Fanuc TP program (LS listing): FM203450.ls

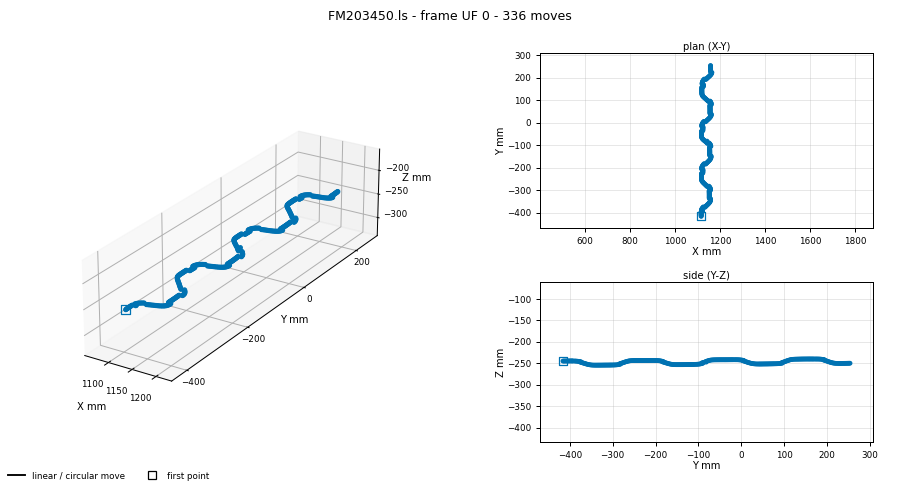
[picture p0: tool path of FM203450.ls in frame UF 0, 336 of 336 moves have a stored position in this frame; points joined in program order, loops and branches not executed]
/PROG  FM203450
/ATTR
OWNER		= MNEDITOR;
COMMENT		= "Auto FANUC move";
PROG_SIZE	= 0;
CREATE		= DATE 26-04-24  TIME 20:34:50;
MODIFIED	= DATE 26-04-24  TIME 20:34:50;
FILE_NAME	= ;
VERSION		= 0;
LINE_COUNT	= 341;
MEMORY_SIZE	= 0;
PROTECT		= READ_WRITE;
TCD:  STACK_SIZE	= 0,
      TASK_PRIORITY	= 50,
      TIME_SLICE	= 0,
      BUSY_LAMP_OFF	= 0,
      ABORT_REQUEST	= 0,
      PAUSE_REQUEST	= 0;
DEFAULT_GROUP	= 1,*,*,*,*;
CONTROL_CODE	= 00000000 00000000;
/MN
   1:  UFRAME_NUM=0 ;
   2:  UTOOL_NUM=1 ;
   3:  R[93]=10 ;
   4:  L P[1] 7mm/sec FINE ;
   5:  L P[2] 7mm/sec CNT50 ;
   6:  L P[3] 7mm/sec CNT50 ;
   7:  L P[4] 7mm/sec CNT50 ;
   8:  L P[5] 7mm/sec CNT50 ;
   9:  L P[6] 7mm/sec CNT50 ;
  10:  L P[7] 7mm/sec CNT50 ;
  11:  L P[8] 7mm/sec CNT50 ;
  12:  L P[9] 7mm/sec CNT50 ;
  13:  L P[10] 7mm/sec CNT50 ;
  14:  L P[11] 7mm/sec CNT50 ;
  15:  L P[12] 7mm/sec CNT50 ;
  16:  L P[13] 7mm/sec CNT50 ;
  17:  L P[14] 7mm/sec CNT50 ;
  18:  L P[15] 7mm/sec CNT50 ;
  19:  L P[16] 7mm/sec CNT50 ;
  20:  L P[17] 7mm/sec CNT50 ;
  21:  L P[18] 7mm/sec CNT50 ;
  22:  L P[19] 7mm/sec CNT50 ;
  23:  L P[20] 7mm/sec CNT50 ;
  24:  L P[21] 7mm/sec CNT50 ;
  25:  L P[22] 7mm/sec CNT50 ;
  26:  L P[23] 7mm/sec CNT50 ;
  27:  L P[24] 7mm/sec CNT50 ;
  28:  L P[25] 7mm/sec CNT50 ;
  29:  L P[26] 7mm/sec CNT50 ;
  30:  L P[27] 7mm/sec CNT50 ;
  31:  L P[28] 7mm/sec CNT50 ;
  32:  L P[29] 7mm/sec CNT50 ;
  33:  L P[30] 7mm/sec CNT50 ;
  34:  L P[31] 7mm/sec CNT50 ;
  35:  L P[32] 7mm/sec CNT50 ;
  36:  L P[33] 7mm/sec CNT50 ;
  37:  L P[34] 7mm/sec CNT50 ;
  38:  L P[35] 7mm/sec CNT50 ;
  39:  L P[36] 7mm/sec CNT50 ;
  40:  L P[37] 7mm/sec CNT50 ;
  41:  L P[38] 7mm/sec CNT50 ;
  42:  L P[39] 7mm/sec CNT50 ;
  43:  L P[40] 7mm/sec CNT50 ;
  44:  L P[41] 7mm/sec CNT50 ;
  45:  L P[42] 7mm/sec CNT50 ;
  46:  L P[43] 7mm/sec CNT50 ;
  47:  L P[44] 7mm/sec CNT50 ;
  48:  L P[45] 7mm/sec CNT50 ;
  49:  L P[46] 7mm/sec CNT50 ;
  50:  L P[47] 7mm/sec CNT50 ;
  51:  L P[48] 7mm/sec CNT50 ;
  52:  L P[49] 7mm/sec CNT50 ;
  53:  L P[50] 7mm/sec CNT50 ;
  54:  L P[51] 7mm/sec CNT50 ;
  55:  L P[52] 7mm/sec CNT50 ;
  56:  L P[53] 7mm/sec CNT50 ;
  57:  L P[54] 7mm/sec CNT50 ;
  58:  L P[55] 7mm/sec CNT50 ;
  59:  L P[56] 7mm/sec CNT50 ;
  60:  L P[57] 7mm/sec CNT50 ;
  61:  L P[58] 7mm/sec CNT50 ;
  62:  L P[59] 7mm/sec CNT50 ;
  63:  L P[60] 7mm/sec CNT50 ;
  64:  L P[61] 7mm/sec CNT50 ;
  65:  L P[62] 7mm/sec CNT50 ;
  66:  L P[63] 7mm/sec CNT50 ;
  67:  L P[64] 7mm/sec CNT50 ;
  68:  L P[65] 7mm/sec CNT50 ;
  69:  L P[66] 7mm/sec CNT50 ;
  70:  L P[67] 7mm/sec CNT50 ;
  71:  L P[68] 7mm/sec CNT50 ;
  72:  L P[69] 7mm/sec CNT50 ;
  73:  L P[70] 7mm/sec CNT50 ;
  74:  L P[71] 7mm/sec CNT50 ;
  75:  L P[72] 7mm/sec CNT50 ;
  76:  L P[73] 7mm/sec CNT50 ;
  77:  L P[74] 7mm/sec CNT50 ;
  78:  L P[75] 7mm/sec CNT50 ;
  79:  L P[76] 7mm/sec CNT50 ;
  80:  L P[77] 7mm/sec CNT50 ;
  81:  L P[78] 7mm/sec CNT50 ;
  82:  L P[79] 7mm/sec CNT50 ;
  83:  L P[80] 7mm/sec CNT50 ;
  84:  L P[81] 7mm/sec CNT50 ;
  85:  L P[82] 7mm/sec CNT50 ;
  86:  L P[83] 7mm/sec CNT50 ;
  87:  L P[84] 7mm/sec CNT50 ;
  88:  L P[85] 7mm/sec CNT50 ;
  89:  L P[86] 7mm/sec CNT50 ;
  90:  L P[87] 7mm/sec CNT50 ;
  91:  L P[88] 7mm/sec CNT50 ;
  92:  L P[89] 7mm/sec CNT50 ;
  93:  L P[90] 7mm/sec CNT50 ;
  94:  L P[91] 7mm/sec CNT50 ;
  95:  L P[92] 7mm/sec CNT50 ;
  96:  L P[93] 7mm/sec CNT50 ;
  97:  L P[94] 7mm/sec CNT50 ;
  98:  L P[95] 7mm/sec CNT50 ;
  99:  L P[96] 7mm/sec CNT50 ;
 100:  L P[97] 7mm/sec CNT50 ;
 101:  L P[98] 7mm/sec CNT50 ;
 102:  L P[99] 7mm/sec CNT50 ;
 103:  L P[100] 7mm/sec CNT50 ;
 104:  L P[101] 7mm/sec CNT50 ;
 105:  L P[102] 7mm/sec CNT50 ;
 106:  L P[103] 7mm/sec CNT50 ;
 107:  L P[104] 7mm/sec CNT50 ;
 108:  L P[105] 7mm/sec CNT50 ;
 109:  L P[106] 7mm/sec CNT50 ;
 110:  L P[107] 7mm/sec CNT50 ;
 111:  L P[108] 7mm/sec CNT50 ;
 112:  L P[109] 7mm/sec CNT50 ;
 113:  L P[110] 7mm/sec CNT50 ;
 114:  L P[111] 7mm/sec CNT50 ;
 115:  L P[112] 7mm/sec CNT50 ;
 116:  L P[113] 7mm/sec CNT50 ;
 117:  L P[114] 7mm/sec CNT50 ;
 118:  L P[115] 7mm/sec CNT50 ;
 119:  L P[116] 7mm/sec CNT50 ;
 120:  L P[117] 7mm/sec CNT50 ;
 121:  L P[118] 7mm/sec CNT50 ;
 122:  L P[119] 7mm/sec CNT50 ;
 123:  L P[120] 7mm/sec CNT50 ;
 124:  L P[121] 7mm/sec CNT50 ;
 125:  L P[122] 7mm/sec CNT50 ;
 126:  L P[123] 7mm/sec CNT50 ;
 127:  L P[124] 7mm/sec CNT50 ;
 128:  L P[125] 7mm/sec CNT50 ;
 129:  L P[126] 7mm/sec CNT50 ;
 130:  L P[127] 7mm/sec CNT50 ;
 131:  L P[128] 7mm/sec CNT50 ;
 132:  L P[129] 7mm/sec CNT50 ;
 133:  L P[130] 7mm/sec CNT50 ;
 134:  L P[131] 7mm/sec CNT50 ;
 135:  L P[132] 7mm/sec CNT50 ;
 136:  L P[133] 7mm/sec CNT50 ;
 137:  L P[134] 7mm/sec CNT50 ;
 138:  L P[135] 7mm/sec CNT50 ;
 139:  L P[136] 7mm/sec CNT50 ;
 140:  L P[137] 7mm/sec CNT50 ;
 141:  L P[138] 7mm/sec CNT50 ;
 142:  L P[139] 7mm/sec CNT50 ;
 143:  L P[140] 7mm/sec CNT50 ;
 144:  L P[141] 7mm/sec CNT50 ;
 145:  L P[142] 7mm/sec CNT50 ;
 146:  L P[143] 7mm/sec CNT50 ;
 147:  L P[144] 7mm/sec CNT50 ;
 148:  L P[145] 7mm/sec CNT50 ;
 149:  L P[146] 7mm/sec CNT50 ;
 150:  L P[147] 7mm/sec CNT50 ;
 151:  L P[148] 7mm/sec CNT50 ;
 152:  L P[149] 7mm/sec CNT50 ;
 153:  L P[150] 7mm/sec CNT50 ;
 154:  L P[151] 7mm/sec CNT50 ;
 155:  L P[152] 7mm/sec CNT50 ;
 156:  L P[153] 7mm/sec CNT50 ;
 157:  L P[154] 7mm/sec CNT50 ;
 158:  L P[155] 7mm/sec CNT50 ;
 159:  L P[156] 7mm/sec CNT50 ;
 160:  L P[157] 7mm/sec CNT50 ;
 161:  L P[158] 7mm/sec CNT50 ;
 162:  L P[159] 7mm/sec CNT50 ;
 163:  L P[160] 7mm/sec CNT50 ;
 164:  L P[161] 7mm/sec CNT50 ;
 165:  L P[162] 7mm/sec CNT50 ;
 166:  L P[163] 7mm/sec CNT50 ;
 167:  L P[164] 7mm/sec CNT50 ;
 168:  L P[165] 7mm/sec CNT50 ;
 169:  L P[166] 7mm/sec CNT50 ;
 170:  L P[167] 7mm/sec CNT50 ;
 171:  L P[168] 7mm/sec CNT50 ;
 172:  L P[169] 7mm/sec CNT50 ;
 173:  L P[170] 7mm/sec CNT50 ;
 174:  L P[171] 7mm/sec CNT50 ;
 175:  L P[172] 7mm/sec CNT50 ;
 176:  L P[173] 7mm/sec CNT50 ;
 177:  L P[174] 7mm/sec CNT50 ;
 178:  L P[175] 7mm/sec CNT50 ;
 179:  L P[176] 7mm/sec CNT50 ;
 180:  L P[177] 7mm/sec CNT50 ;
 181:  L P[178] 7mm/sec CNT50 ;
 182:  L P[179] 7mm/sec CNT50 ;
 183:  L P[180] 7mm/sec CNT50 ;
 184:  L P[181] 7mm/sec CNT50 ;
 185:  L P[182] 7mm/sec CNT50 ;
 186:  L P[183] 7mm/sec CNT50 ;
 187:  L P[184] 7mm/sec CNT50 ;
 188:  L P[185] 7mm/sec CNT50 ;
 189:  L P[186] 7mm/sec CNT50 ;
 190:  L P[187] 7mm/sec CNT50 ;
 191:  L P[188] 7mm/sec CNT50 ;
 192:  L P[189] 7mm/sec CNT50 ;
 193:  L P[190] 7mm/sec CNT50 ;
 194:  L P[191] 7mm/sec CNT50 ;
 195:  L P[192] 7mm/sec CNT50 ;
 196:  L P[193] 7mm/sec CNT50 ;
 197:  L P[194] 7mm/sec CNT50 ;
 198:  L P[195] 7mm/sec CNT50 ;
 199:  L P[196] 7mm/sec CNT50 ;
 200:  L P[197] 7mm/sec CNT50 ;
 201:  L P[198] 7mm/sec CNT50 ;
 202:  L P[199] 7mm/sec CNT50 ;
 203:  L P[200] 7mm/sec CNT50 ;
 204:  L P[201] 7mm/sec CNT50 ;
 205:  L P[202] 7mm/sec CNT50 ;
 206:  L P[203] 7mm/sec CNT50 ;
 207:  L P[204] 7mm/sec CNT50 ;
 208:  L P[205] 7mm/sec CNT50 ;
 209:  L P[206] 7mm/sec CNT50 ;
 210:  L P[207] 7mm/sec CNT50 ;
 211:  L P[208] 7mm/sec CNT50 ;
 212:  L P[209] 7mm/sec CNT50 ;
 213:  L P[210] 7mm/sec CNT50 ;
 214:  L P[211] 7mm/sec CNT50 ;
 215:  L P[212] 7mm/sec CNT50 ;
 216:  L P[213] 7mm/sec CNT50 ;
 217:  L P[214] 7mm/sec CNT50 ;
 218:  L P[215] 7mm/sec CNT50 ;
 219:  L P[216] 7mm/sec CNT50 ;
 220:  L P[217] 7mm/sec CNT50 ;
 221:  L P[218] 7mm/sec CNT50 ;
 222:  L P[219] 7mm/sec CNT50 ;
 223:  L P[220] 7mm/sec CNT50 ;
 224:  L P[221] 7mm/sec CNT50 ;
 225:  L P[222] 7mm/sec CNT50 ;
 226:  L P[223] 7mm/sec CNT50 ;
 227:  L P[224] 7mm/sec CNT50 ;
 228:  L P[225] 7mm/sec CNT50 ;
 229:  L P[226] 7mm/sec CNT50 ;
 230:  L P[227] 7mm/sec CNT50 ;
 231:  L P[228] 7mm/sec CNT50 ;
 232:  L P[229] 7mm/sec CNT50 ;
 233:  L P[230] 7mm/sec CNT50 ;
 234:  L P[231] 7mm/sec CNT50 ;
 235:  L P[232] 7mm/sec CNT50 ;
 236:  L P[233] 7mm/sec CNT50 ;
 237:  L P[234] 7mm/sec CNT50 ;
 238:  L P[235] 7mm/sec CNT50 ;
 239:  L P[236] 7mm/sec CNT50 ;
 240:  L P[237] 7mm/sec CNT50 ;
 241:  L P[238] 7mm/sec CNT50 ;
 242:  L P[239] 7mm/sec CNT50 ;
 243:  L P[240] 7mm/sec CNT50 ;
 244:  L P[241] 7mm/sec CNT50 ;
 245:  L P[242] 7mm/sec CNT50 ;
 246:  L P[243] 7mm/sec CNT50 ;
 247:  L P[244] 7mm/sec CNT50 ;
 248:  L P[245] 7mm/sec CNT50 ;
 249:  L P[246] 7mm/sec CNT50 ;
 250:  L P[247] 7mm/sec CNT50 ;
 251:  L P[248] 7mm/sec CNT50 ;
 252:  L P[249] 7mm/sec CNT50 ;
 253:  L P[250] 7mm/sec CNT50 ;
 254:  L P[251] 7mm/sec CNT50 ;
 255:  L P[252] 7mm/sec CNT50 ;
 256:  L P[253] 7mm/sec CNT50 ;
 257:  L P[254] 7mm/sec CNT50 ;
 258:  L P[255] 7mm/sec CNT50 ;
 259:  L P[256] 7mm/sec CNT50 ;
 260:  L P[257] 7mm/sec CNT50 ;
 261:  L P[258] 7mm/sec CNT50 ;
 262:  L P[259] 7mm/sec CNT50 ;
 263:  L P[260] 7mm/sec CNT50 ;
 264:  L P[261] 7mm/sec CNT50 ;
 265:  L P[262] 7mm/sec CNT50 ;
 266:  L P[263] 7mm/sec CNT50 ;
 267:  L P[264] 7mm/sec CNT50 ;
 268:  L P[265] 7mm/sec CNT50 ;
 269:  L P[266] 7mm/sec CNT50 ;
 270:  L P[267] 7mm/sec CNT50 ;
 271:  L P[268] 7mm/sec CNT50 ;
 272:  L P[269] 7mm/sec CNT50 ;
 273:  L P[270] 7mm/sec CNT50 ;
 274:  L P[271] 7mm/sec CNT50 ;
 275:  L P[272] 7mm/sec CNT50 ;
 276:  L P[273] 7mm/sec CNT50 ;
 277:  L P[274] 7mm/sec CNT50 ;
 278:  L P[275] 7mm/sec CNT50 ;
 279:  L P[276] 7mm/sec CNT50 ;
 280:  L P[277] 7mm/sec CNT50 ;
 281:  L P[278] 7mm/sec CNT50 ;
 282:  L P[279] 7mm/sec CNT50 ;
 283:  L P[280] 7mm/sec CNT50 ;
 284:  L P[281] 7mm/sec CNT50 ;
 285:  L P[282] 7mm/sec CNT50 ;
 286:  L P[283] 7mm/sec CNT50 ;
 287:  L P[284] 7mm/sec CNT50 ;
 288:  L P[285] 7mm/sec CNT50 ;
 289:  L P[286] 7mm/sec CNT50 ;
 290:  L P[287] 7mm/sec CNT50 ;
 291:  L P[288] 7mm/sec CNT50 ;
 292:  L P[289] 7mm/sec CNT50 ;
 293:  L P[290] 7mm/sec CNT50 ;
 294:  L P[291] 7mm/sec CNT50 ;
 295:  L P[292] 7mm/sec CNT50 ;
 296:  L P[293] 7mm/sec CNT50 ;
 297:  L P[294] 7mm/sec CNT50 ;
 298:  L P[295] 7mm/sec CNT50 ;
 299:  L P[296] 7mm/sec CNT50 ;
 300:  L P[297] 7mm/sec CNT50 ;
 301:  L P[298] 7mm/sec CNT50 ;
 302:  L P[299] 7mm/sec CNT50 ;
 303:  L P[300] 7mm/sec CNT50 ;
 304:  L P[301] 7mm/sec CNT50 ;
 305:  L P[302] 7mm/sec CNT50 ;
 306:  L P[303] 7mm/sec CNT50 ;
 307:  L P[304] 7mm/sec CNT50 ;
 308:  L P[305] 7mm/sec CNT50 ;
 309:  L P[306] 7mm/sec CNT50 ;
 310:  L P[307] 7mm/sec CNT50 ;
 311:  L P[308] 7mm/sec CNT50 ;
 312:  L P[309] 7mm/sec CNT50 ;
 313:  L P[310] 7mm/sec CNT50 ;
 314:  L P[311] 7mm/sec CNT50 ;
 315:  L P[312] 7mm/sec CNT50 ;
 316:  L P[313] 7mm/sec CNT50 ;
 317:  L P[314] 7mm/sec CNT50 ;
 318:  L P[315] 7mm/sec CNT50 ;
 319:  L P[316] 7mm/sec CNT50 ;
 320:  L P[317] 7mm/sec CNT50 ;
 321:  L P[318] 7mm/sec CNT50 ;
 322:  L P[319] 7mm/sec CNT50 ;
 323:  L P[320] 7mm/sec CNT50 ;
 324:  L P[321] 7mm/sec CNT50 ;
 325:  L P[322] 7mm/sec CNT50 ;
 326:  L P[323] 7mm/sec CNT50 ;
 327:  L P[324] 7mm/sec CNT50 ;
 328:  L P[325] 7mm/sec CNT50 ;
 329:  L P[326] 7mm/sec CNT50 ;
 330:  L P[327] 7mm/sec CNT50 ;
 331:  L P[328] 7mm/sec CNT50 ;
 332:  L P[329] 7mm/sec CNT50 ;
 333:  L P[330] 7mm/sec CNT50 ;
 334:  L P[331] 7mm/sec CNT50 ;
 335:  L P[332] 7mm/sec CNT50 ;
 336:  L P[333] 7mm/sec CNT50 ;
 337:  L P[334] 7mm/sec CNT50 ;
 338:  L P[335] 7mm/sec CNT50 ;
 339:  L P[336] 7mm/sec FINE ;
 340:  R[93]=1 ;
 341:  END ;
/POS
P[1]{
   GP1:
	UF : 0, UT : 1,		CONFIG : 'N U T, 0, 0, 0',
	X = 1117.238  mm,	Y = -416.121  mm,	Z = -244.812  mm,
	W = 0.000 deg,	P = 30.000 deg,	R = 175.456 deg
};
P[2]{
   GP1:
	UF : 0, UT : 1,		CONFIG : 'N U T, 0, 0, 0',
	X = 1117.157  mm,	Y = -414.122  mm,	Z = -244.780  mm,
	W = 0.000 deg,	P = 30.000 deg,	R = 175.456 deg
};
P[3]{
   GP1:
	UF : 0, UT : 1,		CONFIG : 'N U T, 0, 0, 0',
	X = 1117.075  mm,	Y = -412.113  mm,	Z = -244.742  mm,
	W = 0.000 deg,	P = 30.000 deg,	R = 175.456 deg
};
P[4]{
   GP1:
	UF : 0, UT : 1,		CONFIG : 'N U T, 0, 0, 0',
	X = 1117.006  mm,	Y = -410.100  mm,	Z = -244.707  mm,
	W = 0.000 deg,	P = 30.000 deg,	R = 175.456 deg
};
P[5]{
   GP1:
	UF : 0, UT : 1,		CONFIG : 'N U T, 0, 0, 0',
	X = 1116.940  mm,	Y = -408.081  mm,	Z = -244.666  mm,
	W = 0.000 deg,	P = 30.000 deg,	R = 175.456 deg
};
P[6]{
   GP1:
	UF : 0, UT : 1,		CONFIG : 'N U T, 0, 0, 0',
	X = 1116.897  mm,	Y = -406.053  mm,	Z = -244.628  mm,
	W = 0.000 deg,	P = 30.000 deg,	R = 175.456 deg
};
P[7]{
   GP1:
	UF : 0, UT : 1,		CONFIG : 'N U T, 0, 0, 0',
	X = 1116.868  mm,	Y = -404.029  mm,	Z = -244.597  mm,
	W = 0.000 deg,	P = 30.000 deg,	R = 175.456 deg
};
P[8]{
   GP1:
	UF : 0, UT : 1,		CONFIG : 'N U T, 0, 0, 0',
	X = 1116.858  mm,	Y = -402.004  mm,	Z = -244.573  mm,
	W = 0.000 deg,	P = 30.000 deg,	R = 175.456 deg
};
P[9]{
   GP1:
	UF : 0, UT : 1,		CONFIG : 'N U T, 0, 0, 0',
	X = 1116.863  mm,	Y = -399.971  mm,	Z = -244.558  mm,
	W = 0.000 deg,	P = 30.000 deg,	R = 175.456 deg
};
P[10]{
   GP1:
	UF : 0, UT : 1,		CONFIG : 'N U T, 0, 0, 0',
	X = 1116.898  mm,	Y = -397.917  mm,	Z = -244.550  mm,
	W = 0.000 deg,	P = 30.000 deg,	R = 175.456 deg
};
P[11]{
   GP1:
	UF : 0, UT : 1,		CONFIG : 'N U T, 0, 0, 0',
	X = 1116.977  mm,	Y = -395.859  mm,	Z = -244.552  mm,
	W = 0.000 deg,	P = 30.000 deg,	R = 175.456 deg
};
P[12]{
   GP1:
	UF : 0, UT : 1,		CONFIG : 'N U T, 0, 0, 0',
	X = 1123.071  mm,	Y = -394.287  mm,	Z = -244.568  mm,
	W = 0.000 deg,	P = 30.000 deg,	R = 175.456 deg
};
P[13]{
   GP1:
	UF : 0, UT : 1,		CONFIG : 'N U T, 0, 0, 0',
	X = 1123.311  mm,	Y = -392.534  mm,	Z = -244.620  mm,
	W = 0.000 deg,	P = 30.000 deg,	R = 170.071 deg
};
P[14]{
   GP1:
	UF : 0, UT : 1,		CONFIG : 'N U T, 0, 0, 0',
	X = 1117.902  mm,	Y = -389.257  mm,	Z = -244.722  mm,
	W = 0.000 deg,	P = 30.000 deg,	R = 162.234 deg
};
P[15]{
   GP1:
	UF : 0, UT : 1,		CONFIG : 'N U T, 0, 0, 0',
	X = 1118.551  mm,	Y = -387.006  mm,	Z = -244.847  mm,
	W = 0.000 deg,	P = 30.000 deg,	R = 154.276 deg
};
P[16]{
   GP1:
	UF : 0, UT : 1,		CONFIG : 'N U T, 0, 0, 0',
	X = 1119.505  mm,	Y = -384.707  mm,	Z = -245.002  mm,
	W = 0.000 deg,	P = 30.000 deg,	R = 145.985 deg
};
P[17]{
   GP1:
	UF : 0, UT : 1,		CONFIG : 'N U T, 0, 0, 0',
	X = 1120.698  mm,	Y = -382.492  mm,	Z = -245.205  mm,
	W = 0.000 deg,	P = 30.000 deg,	R = 137.274 deg
};
P[18]{
   GP1:
	UF : 0, UT : 1,		CONFIG : 'N U T, 0, 0, 0',
	X = 1122.055  mm,	Y = -380.317  mm,	Z = -245.479  mm,
	W = 0.000 deg,	P = 30.000 deg,	R = 137.274 deg
};
P[19]{
   GP1:
	UF : 0, UT : 1,		CONFIG : 'N U T, 0, 0, 0',
	X = 1123.594  mm,	Y = -378.210  mm,	Z = -245.828  mm,
	W = 0.000 deg,	P = 30.000 deg,	R = 137.274 deg
};
P[20]{
   GP1:
	UF : 0, UT : 1,		CONFIG : 'N U T, 0, 0, 0',
	X = 1125.169  mm,	Y = -376.126  mm,	Z = -246.227  mm,
	W = 0.000 deg,	P = 30.000 deg,	R = 137.274 deg
};
P[21]{
   GP1:
	UF : 0, UT : 1,		CONFIG : 'N U T, 0, 0, 0',
	X = 1126.962  mm,	Y = -374.005  mm,	Z = -246.664  mm,
	W = 0.000 deg,	P = 30.000 deg,	R = 137.274 deg
};
P[22]{
   GP1:
	UF : 0, UT : 1,		CONFIG : 'N U T, 0, 0, 0',
	X = 1133.263  mm,	Y = -376.051  mm,	Z = -247.177  mm,
	W = 0.000 deg,	P = 30.000 deg,	R = 137.274 deg
};
P[23]{
   GP1:
	UF : 0, UT : 1,		CONFIG : 'N U T, 0, 0, 0',
	X = 1135.120  mm,	Y = -374.071  mm,	Z = -247.739  mm,
	W = 0.000 deg,	P = 30.000 deg,	R = 137.274 deg
};
P[24]{
   GP1:
	UF : 0, UT : 1,		CONFIG : 'N U T, 0, 0, 0',
	X = 1137.025  mm,	Y = -372.109  mm,	Z = -248.355  mm,
	W = 0.000 deg,	P = 30.000 deg,	R = 137.274 deg
};
P[25]{
   GP1:
	UF : 0, UT : 1,		CONFIG : 'N U T, 0, 0, 0',
	X = 1138.998  mm,	Y = -370.148  mm,	Z = -248.981  mm,
	W = 0.000 deg,	P = 30.000 deg,	R = 137.274 deg
};
P[26]{
   GP1:
	UF : 0, UT : 1,		CONFIG : 'N U T, 0, 0, 0',
	X = 1141.067  mm,	Y = -368.170  mm,	Z = -249.617  mm,
	W = 0.000 deg,	P = 30.000 deg,	R = 137.274 deg
};
P[27]{
   GP1:
	UF : 0, UT : 1,		CONFIG : 'N U T, 0, 0, 0',
	X = 1143.185  mm,	Y = -366.152  mm,	Z = -250.236  mm,
	W = 0.000 deg,	P = 30.000 deg,	R = 137.274 deg
};
P[28]{
   GP1:
	UF : 0, UT : 1,		CONFIG : 'N U T, 0, 0, 0',
	X = 1145.220  mm,	Y = -364.138  mm,	Z = -250.854  mm,
	W = 0.000 deg,	P = 30.000 deg,	R = 137.274 deg
};
P[29]{
   GP1:
	UF : 0, UT : 1,		CONFIG : 'N U T, 0, 0, 0',
	X = 1147.260  mm,	Y = -362.140  mm,	Z = -251.461  mm,
	W = 0.000 deg,	P = 30.000 deg,	R = 143.931 deg
};
P[30]{
   GP1:
	UF : 0, UT : 1,		CONFIG : 'N U T, 0, 0, 0',
	X = 1149.327  mm,	Y = -360.100  mm,	Z = -252.059  mm,
	W = 0.000 deg,	P = 30.000 deg,	R = 156.053 deg
};
P[31]{
   GP1:
	UF : 0, UT : 1,		CONFIG : 'N U T, 0, 0, 0',
	X = 1151.305  mm,	Y = -358.012  mm,	Z = -252.604  mm,
	W = 0.000 deg,	P = 30.000 deg,	R = 167.750 deg
};
P[32]{
   GP1:
	UF : 0, UT : 1,		CONFIG : 'N U T, 0, 0, 0',
	X = 1153.153  mm,	Y = -355.863  mm,	Z = -253.093  mm,
	W = 0.000 deg,	P = 30.000 deg,	R = 178.930 deg
};
P[33]{
   GP1:
	UF : 0, UT : 1,		CONFIG : 'N U T, 0, 0, 0',
	X = 1154.738  mm,	Y = -353.672  mm,	Z = -253.493  mm,
	W = 0.000 deg,	P = 30.000 deg,	R = 178.930 deg
};
P[34]{
   GP1:
	UF : 0, UT : 1,		CONFIG : 'N U T, 0, 0, 0',
	X = 1156.111  mm,	Y = -351.454  mm,	Z = -253.825  mm,
	W = 0.000 deg,	P = 30.000 deg,	R = 178.930 deg
};
P[35]{
   GP1:
	UF : 0, UT : 1,		CONFIG : 'N U T, 0, 0, 0',
	X = 1157.241  mm,	Y = -349.136  mm,	Z = -254.072  mm,
	W = 0.000 deg,	P = 30.000 deg,	R = 178.930 deg
};
P[36]{
   GP1:
	UF : 0, UT : 1,		CONFIG : 'N U T, 0, 0, 0',
	X = 1158.022  mm,	Y = -346.774  mm,	Z = -254.230  mm,
	W = 0.000 deg,	P = 30.000 deg,	R = 178.930 deg
};
P[37]{
   GP1:
	UF : 0, UT : 1,		CONFIG : 'N U T, 0, 0, 0',
	X = 1158.497  mm,	Y = -344.458  mm,	Z = -254.317  mm,
	W = 0.000 deg,	P = 30.000 deg,	R = 178.930 deg
};
P[38]{
   GP1:
	UF : 0, UT : 1,		CONFIG : 'N U T, 0, 0, 0',
	X = 1158.732  mm,	Y = -342.235  mm,	Z = -254.352  mm,
	W = 0.000 deg,	P = 30.000 deg,	R = 178.930 deg
};
P[39]{
   GP1:
	UF : 0, UT : 1,		CONFIG : 'N U T, 0, 0, 0',
	X = 1158.843  mm,	Y = -340.119  mm,	Z = -254.355  mm,
	W = 0.000 deg,	P = 30.000 deg,	R = 178.930 deg
};
P[40]{
   GP1:
	UF : 0, UT : 1,		CONFIG : 'N U T, 0, 0, 0',
	X = 1158.899  mm,	Y = -338.073  mm,	Z = -254.354  mm,
	W = 0.000 deg,	P = 30.000 deg,	R = 178.930 deg
};
P[41]{
   GP1:
	UF : 0, UT : 1,		CONFIG : 'N U T, 0, 0, 0',
	X = 1152.944  mm,	Y = -335.946  mm,	Z = -254.352  mm,
	W = 0.000 deg,	P = 30.000 deg,	R = 178.930 deg
};
P[42]{
   GP1:
	UF : 0, UT : 1,		CONFIG : 'N U T, 0, 0, 0',
	X = 1152.971  mm,	Y = -333.966  mm,	Z = -254.346  mm,
	W = 0.000 deg,	P = 30.000 deg,	R = 178.930 deg
};
P[43]{
   GP1:
	UF : 0, UT : 1,		CONFIG : 'N U T, 0, 0, 0',
	X = 1152.989  mm,	Y = -331.976  mm,	Z = -254.338  mm,
	W = 0.000 deg,	P = 30.000 deg,	R = 178.930 deg
};
P[44]{
   GP1:
	UF : 0, UT : 1,		CONFIG : 'N U T, 0, 0, 0',
	X = 1153.003  mm,	Y = -329.982  mm,	Z = -254.324  mm,
	W = 0.000 deg,	P = 30.000 deg,	R = 178.930 deg
};
P[45]{
   GP1:
	UF : 0, UT : 1,		CONFIG : 'N U T, 0, 0, 0',
	X = 1153.013  mm,	Y = -327.989  mm,	Z = -254.307  mm,
	W = 0.000 deg,	P = 30.000 deg,	R = 178.930 deg
};
P[46]{
   GP1:
	UF : 0, UT : 1,		CONFIG : 'N U T, 0, 0, 0',
	X = 1153.018  mm,	Y = -325.995  mm,	Z = -254.288  mm,
	W = 0.000 deg,	P = 30.000 deg,	R = 178.930 deg
};
P[47]{
   GP1:
	UF : 0, UT : 1,		CONFIG : 'N U T, 0, 0, 0',
	X = 1153.020  mm,	Y = -323.998  mm,	Z = -254.268  mm,
	W = 0.000 deg,	P = 30.000 deg,	R = 178.930 deg
};
P[48]{
   GP1:
	UF : 0, UT : 1,		CONFIG : 'N U T, 0, 0, 0',
	X = 1153.020  mm,	Y = -322.002  mm,	Z = -254.247  mm,
	W = 0.000 deg,	P = 30.000 deg,	R = 178.930 deg
};
P[49]{
   GP1:
	UF : 0, UT : 1,		CONFIG : 'N U T, 0, 0, 0',
	X = 1153.017  mm,	Y = -320.009  mm,	Z = -254.228  mm,
	W = 0.000 deg,	P = 30.000 deg,	R = 178.930 deg
};
P[50]{
   GP1:
	UF : 0, UT : 1,		CONFIG : 'N U T, 0, 0, 0',
	X = 1153.008  mm,	Y = -318.019  mm,	Z = -254.209  mm,
	W = 0.000 deg,	P = 30.000 deg,	R = 178.930 deg
};
P[51]{
   GP1:
	UF : 0, UT : 1,		CONFIG : 'N U T, 0, 0, 0',
	X = 1152.993  mm,	Y = -316.026  mm,	Z = -254.195  mm,
	W = 0.000 deg,	P = 30.000 deg,	R = 178.930 deg
};
P[52]{
   GP1:
	UF : 0, UT : 1,		CONFIG : 'N U T, 0, 0, 0',
	X = 1152.973  mm,	Y = -314.036  mm,	Z = -254.181  mm,
	W = 0.000 deg,	P = 30.000 deg,	R = 178.930 deg
};
P[53]{
   GP1:
	UF : 0, UT : 1,		CONFIG : 'N U T, 0, 0, 0',
	X = 1152.945  mm,	Y = -312.050  mm,	Z = -254.166  mm,
	W = 0.000 deg,	P = 30.000 deg,	R = 178.930 deg
};
P[54]{
   GP1:
	UF : 0, UT : 1,		CONFIG : 'N U T, 0, 0, 0',
	X = 1152.907  mm,	Y = -310.067  mm,	Z = -254.149  mm,
	W = 0.000 deg,	P = 30.000 deg,	R = 178.930 deg
};
P[55]{
   GP1:
	UF : 0, UT : 1,		CONFIG : 'N U T, 0, 0, 0',
	X = 1152.856  mm,	Y = -308.083  mm,	Z = -254.127  mm,
	W = 0.000 deg,	P = 30.000 deg,	R = 178.930 deg
};
P[56]{
   GP1:
	UF : 0, UT : 1,		CONFIG : 'N U T, 0, 0, 0',
	X = 1152.797  mm,	Y = -306.094  mm,	Z = -254.104  mm,
	W = 0.000 deg,	P = 30.000 deg,	R = 178.930 deg
};
P[57]{
   GP1:
	UF : 0, UT : 1,		CONFIG : 'N U T, 0, 0, 0',
	X = 1152.731  mm,	Y = -304.105  mm,	Z = -254.075  mm,
	W = 0.000 deg,	P = 30.000 deg,	R = 178.930 deg
};
P[58]{
   GP1:
	UF : 0, UT : 1,		CONFIG : 'N U T, 0, 0, 0',
	X = 1152.659  mm,	Y = -302.140  mm,	Z = -254.045  mm,
	W = 0.000 deg,	P = 30.000 deg,	R = 178.930 deg
};
P[59]{
   GP1:
	UF : 0, UT : 1,		CONFIG : 'N U T, 0, 0, 0',
	X = 1158.536  mm,	Y = -299.819  mm,	Z = -253.999  mm,
	W = 0.000 deg,	P = 30.000 deg,	R = -172.792 deg
};
P[60]{
   GP1:
	UF : 0, UT : 1,		CONFIG : 'N U T, 0, 0, 0',
	X = 1158.403  mm,	Y = -297.754  mm,	Z = -253.948  mm,
	W = 0.000 deg,	P = 30.000 deg,	R = -163.956 deg
};
P[61]{
   GP1:
	UF : 0, UT : 1,		CONFIG : 'N U T, 0, 0, 0',
	X = 1158.189  mm,	Y = -295.627  mm,	Z = -253.878  mm,
	W = 0.000 deg,	P = 30.000 deg,	R = -155.091 deg
};
P[62]{
   GP1:
	UF : 0, UT : 1,		CONFIG : 'N U T, 0, 0, 0',
	X = 1157.847  mm,	Y = -293.378  mm,	Z = -253.781  mm,
	W = 0.000 deg,	P = 30.000 deg,	R = -146.168 deg
};
P[63]{
   GP1:
	UF : 0, UT : 1,		CONFIG : 'N U T, 0, 0, 0',
	X = 1157.172  mm,	Y = -290.942  mm,	Z = -253.605  mm,
	W = 0.000 deg,	P = 30.000 deg,	R = -136.996 deg
};
P[64]{
   GP1:
	UF : 0, UT : 1,		CONFIG : 'N U T, 0, 0, 0',
	X = 1156.021  mm,	Y = -288.532  mm,	Z = -253.312  mm,
	W = 0.000 deg,	P = 30.000 deg,	R = -136.996 deg
};
P[65]{
   GP1:
	UF : 0, UT : 1,		CONFIG : 'N U T, 0, 0, 0',
	X = 1154.591  mm,	Y = -286.300  mm,	Z = -252.918  mm,
	W = 0.000 deg,	P = 30.000 deg,	R = -136.996 deg
};
P[66]{
   GP1:
	UF : 0, UT : 1,		CONFIG : 'N U T, 0, 0, 0',
	X = 1152.986  mm,	Y = -284.113  mm,	Z = -252.468  mm,
	W = 0.000 deg,	P = 30.000 deg,	R = -136.996 deg
};
P[67]{
   GP1:
	UF : 0, UT : 1,		CONFIG : 'N U T, 0, 0, 0',
	X = 1151.105  mm,	Y = -281.983  mm,	Z = -251.928  mm,
	W = 0.000 deg,	P = 30.000 deg,	R = -136.996 deg
};
P[68]{
   GP1:
	UF : 0, UT : 1,		CONFIG : 'N U T, 0, 0, 0',
	X = 1144.899  mm,	Y = -284.123  mm,	Z = -251.352  mm,
	W = 0.000 deg,	P = 30.000 deg,	R = -136.996 deg
};
P[69]{
   GP1:
	UF : 0, UT : 1,		CONFIG : 'N U T, 0, 0, 0',
	X = 1142.839  mm,	Y = -282.199  mm,	Z = -250.685  mm,
	W = 0.000 deg,	P = 30.000 deg,	R = -136.996 deg
};
P[70]{
   GP1:
	UF : 0, UT : 1,		CONFIG : 'N U T, 0, 0, 0',
	X = 1140.618  mm,	Y = -280.151  mm,	Z = -250.008  mm,
	W = 0.000 deg,	P = 30.000 deg,	R = -136.996 deg
};
P[71]{
   GP1:
	UF : 0, UT : 1,		CONFIG : 'N U T, 0, 0, 0',
	X = 1138.641  mm,	Y = -278.119  mm,	Z = -249.386  mm,
	W = 0.000 deg,	P = 30.000 deg,	R = -136.996 deg
};
P[72]{
   GP1:
	UF : 0, UT : 1,		CONFIG : 'N U T, 0, 0, 0',
	X = 1136.600  mm,	Y = -276.125  mm,	Z = -248.711  mm,
	W = 0.000 deg,	P = 30.000 deg,	R = -136.996 deg
};
P[73]{
   GP1:
	UF : 0, UT : 1,		CONFIG : 'N U T, 0, 0, 0',
	X = 1134.609  mm,	Y = -274.102  mm,	Z = -248.054  mm,
	W = 0.000 deg,	P = 30.000 deg,	R = -136.996 deg
};
P[74]{
   GP1:
	UF : 0, UT : 1,		CONFIG : 'N U T, 0, 0, 0',
	X = 1132.747  mm,	Y = -272.196  mm,	Z = -247.379  mm,
	W = 0.000 deg,	P = 30.000 deg,	R = -136.996 deg
};
P[75]{
   GP1:
	UF : 0, UT : 1,		CONFIG : 'N U T, 0, 0, 0',
	X = 1130.424  mm,	Y = -270.212  mm,	Z = -246.656  mm,
	W = 0.000 deg,	P = 30.000 deg,	R = -136.996 deg
};
P[76]{
   GP1:
	UF : 0, UT : 1,		CONFIG : 'N U T, 0, 0, 0',
	X = 1128.315  mm,	Y = -268.134  mm,	Z = -246.043  mm,
	W = 0.000 deg,	P = 30.000 deg,	R = -144.486 deg
};
P[77]{
   GP1:
	UF : 0, UT : 1,		CONFIG : 'N U T, 0, 0, 0',
	X = 1126.263  mm,	Y = -266.105  mm,	Z = -245.449  mm,
	W = 0.000 deg,	P = 30.000 deg,	R = -157.136 deg
};
P[78]{
   GP1:
	UF : 0, UT : 1,		CONFIG : 'N U T, 0, 0, 0',
	X = 1124.213  mm,	Y = -263.958  mm,	Z = -244.899  mm,
	W = 0.000 deg,	P = 30.000 deg,	R = -169.430 deg
};
P[79]{
   GP1:
	UF : 0, UT : 1,		CONFIG : 'N U T, 0, 0, 0',
	X = 1122.535  mm,	Y = -261.771  mm,	Z = -244.489  mm,
	W = 0.000 deg,	P = 30.000 deg,	R = 179.462 deg
};
P[80]{
   GP1:
	UF : 0, UT : 1,		CONFIG : 'N U T, 0, 0, 0',
	X = 1121.010  mm,	Y = -259.579  mm,	Z = -244.131  mm,
	W = 0.000 deg,	P = 30.000 deg,	R = 179.462 deg
};
P[81]{
   GP1:
	UF : 0, UT : 1,		CONFIG : 'N U T, 0, 0, 0',
	X = 1119.695  mm,	Y = -257.117  mm,	Z = -243.885  mm,
	W = 0.000 deg,	P = 30.000 deg,	R = 179.462 deg
};
P[82]{
   GP1:
	UF : 0, UT : 1,		CONFIG : 'N U T, 0, 0, 0',
	X = 1119.040  mm,	Y = -254.711  mm,	Z = -243.744  mm,
	W = 0.000 deg,	P = 30.000 deg,	R = 179.462 deg
};
P[83]{
   GP1:
	UF : 0, UT : 1,		CONFIG : 'N U T, 0, 0, 0',
	X = 1118.539  mm,	Y = -252.460  mm,	Z = -243.614  mm,
	W = 0.000 deg,	P = 30.000 deg,	R = 179.462 deg
};
P[84]{
   GP1:
	UF : 0, UT : 1,		CONFIG : 'N U T, 0, 0, 0',
	X = 1118.340  mm,	Y = -250.184  mm,	Z = -243.552  mm,
	W = 0.000 deg,	P = 30.000 deg,	R = 179.462 deg
};
P[85]{
   GP1:
	UF : 0, UT : 1,		CONFIG : 'N U T, 0, 0, 0',
	X = 1118.258  mm,	Y = -248.073  mm,	Z = -243.512  mm,
	W = 0.000 deg,	P = 30.000 deg,	R = 179.462 deg
};
P[86]{
   GP1:
	UF : 0, UT : 1,		CONFIG : 'N U T, 0, 0, 0',
	X = 1118.238  mm,	Y = -246.020  mm,	Z = -243.487  mm,
	W = 0.000 deg,	P = 30.000 deg,	R = 179.462 deg
};
P[87]{
   GP1:
	UF : 0, UT : 1,		CONFIG : 'N U T, 0, 0, 0',
	X = 1118.231  mm,	Y = -244.007  mm,	Z = -243.465  mm,
	W = 0.000 deg,	P = 30.000 deg,	R = 179.462 deg
};
P[88]{
   GP1:
	UF : 0, UT : 1,		CONFIG : 'N U T, 0, 0, 0',
	X = 1118.229  mm,	Y = -242.001  mm,	Z = -243.446  mm,
	W = 0.000 deg,	P = 30.000 deg,	R = 179.462 deg
};
P[89]{
   GP1:
	UF : 0, UT : 1,		CONFIG : 'N U T, 0, 0, 0',
	X = 1118.229  mm,	Y = -239.998  mm,	Z = -243.428  mm,
	W = 0.000 deg,	P = 30.000 deg,	R = 179.462 deg
};
P[90]{
   GP1:
	UF : 0, UT : 1,		CONFIG : 'N U T, 0, 0, 0',
	X = 1118.231  mm,	Y = -237.996  mm,	Z = -243.411  mm,
	W = 0.000 deg,	P = 30.000 deg,	R = 179.462 deg
};
P[91]{
   GP1:
	UF : 0, UT : 1,		CONFIG : 'N U T, 0, 0, 0',
	X = 1118.234  mm,	Y = -235.995  mm,	Z = -243.397  mm,
	W = 0.000 deg,	P = 30.000 deg,	R = 179.462 deg
};
P[92]{
   GP1:
	UF : 0, UT : 1,		CONFIG : 'N U T, 0, 0, 0',
	X = 1118.238  mm,	Y = -233.995  mm,	Z = -243.388  mm,
	W = 0.000 deg,	P = 30.000 deg,	R = 179.462 deg
};
P[93]{
   GP1:
	UF : 0, UT : 1,		CONFIG : 'N U T, 0, 0, 0',
	X = 1118.241  mm,	Y = -231.994  mm,	Z = -243.377  mm,
	W = 0.000 deg,	P = 30.000 deg,	R = 179.462 deg
};
P[94]{
   GP1:
	UF : 0, UT : 1,		CONFIG : 'N U T, 0, 0, 0',
	X = 1118.245  mm,	Y = -229.992  mm,	Z = -243.366  mm,
	W = 0.000 deg,	P = 30.000 deg,	R = 179.462 deg
};
P[95]{
   GP1:
	UF : 0, UT : 1,		CONFIG : 'N U T, 0, 0, 0',
	X = 1118.252  mm,	Y = -227.987  mm,	Z = -243.356  mm,
	W = 0.000 deg,	P = 30.000 deg,	R = 179.462 deg
};
P[96]{
   GP1:
	UF : 0, UT : 1,		CONFIG : 'N U T, 0, 0, 0',
	X = 1118.262  mm,	Y = -225.976  mm,	Z = -243.347  mm,
	W = 0.000 deg,	P = 30.000 deg,	R = 179.462 deg
};
P[97]{
   GP1:
	UF : 0, UT : 1,		CONFIG : 'N U T, 0, 0, 0',
	X = 1124.284  mm,	Y = -224.034  mm,	Z = -243.337  mm,
	W = 0.000 deg,	P = 30.000 deg,	R = 179.462 deg
};
P[98]{
   GP1:
	UF : 0, UT : 1,		CONFIG : 'N U T, 0, 0, 0',
	X = 1124.308  mm,	Y = -222.043  mm,	Z = -243.327  mm,
	W = 0.000 deg,	P = 30.000 deg,	R = 179.462 deg
};
P[99]{
   GP1:
	UF : 0, UT : 1,		CONFIG : 'N U T, 0, 0, 0',
	X = 1124.341  mm,	Y = -220.057  mm,	Z = -243.317  mm,
	W = 0.000 deg,	P = 30.000 deg,	R = 179.462 deg
};
P[100]{
   GP1:
	UF : 0, UT : 1,		CONFIG : 'N U T, 0, 0, 0',
	X = 1124.383  mm,	Y = -218.070  mm,	Z = -243.307  mm,
	W = 0.000 deg,	P = 30.000 deg,	R = 179.462 deg
};
P[101]{
   GP1:
	UF : 0, UT : 1,		CONFIG : 'N U T, 0, 0, 0',
	X = 1124.434  mm,	Y = -216.086  mm,	Z = -243.300  mm,
	W = 0.000 deg,	P = 30.000 deg,	R = 179.462 deg
};
P[102]{
   GP1:
	UF : 0, UT : 1,		CONFIG : 'N U T, 0, 0, 0',
	X = 1124.497  mm,	Y = -214.108  mm,	Z = -243.294  mm,
	W = 0.000 deg,	P = 30.000 deg,	R = 179.462 deg
};
P[103]{
   GP1:
	UF : 0, UT : 1,		CONFIG : 'N U T, 0, 0, 0',
	X = 1124.577  mm,	Y = -212.127  mm,	Z = -243.289  mm,
	W = 0.000 deg,	P = 30.000 deg,	R = 179.462 deg
};
P[104]{
   GP1:
	UF : 0, UT : 1,		CONFIG : 'N U T, 0, 0, 0',
	X = 1124.665  mm,	Y = -210.153  mm,	Z = -243.289  mm,
	W = 0.000 deg,	P = 30.000 deg,	R = 179.462 deg
};
P[105]{
   GP1:
	UF : 0, UT : 1,		CONFIG : 'N U T, 0, 0, 0',
	X = 1124.778  mm,	Y = -208.184  mm,	Z = -243.293  mm,
	W = 0.000 deg,	P = 30.000 deg,	R = 179.462 deg
};
P[106]{
   GP1:
	UF : 0, UT : 1,		CONFIG : 'N U T, 0, 0, 0',
	X = 1118.923  mm,	Y = -205.767  mm,	Z = -243.301  mm,
	W = 0.000 deg,	P = 30.000 deg,	R = 171.909 deg
};
P[107]{
   GP1:
	UF : 0, UT : 1,		CONFIG : 'N U T, 0, 0, 0',
	X = 1119.114  mm,	Y = -203.661  mm,	Z = -243.323  mm,
	W = 0.000 deg,	P = 30.000 deg,	R = 163.696 deg
};
P[108]{
   GP1:
	UF : 0, UT : 1,		CONFIG : 'N U T, 0, 0, 0',
	X = 1119.409  mm,	Y = -201.512  mm,	Z = -243.366  mm,
	W = 0.000 deg,	P = 30.000 deg,	R = 155.438 deg
};
P[109]{
   GP1:
	UF : 0, UT : 1,		CONFIG : 'N U T, 0, 0, 0',
	X = 1119.838  mm,	Y = -199.293  mm,	Z = -243.440  mm,
	W = 0.000 deg,	P = 30.000 deg,	R = 147.103 deg
};
P[110]{
   GP1:
	UF : 0, UT : 1,		CONFIG : 'N U T, 0, 0, 0',
	X = 1120.504  mm,	Y = -197.016  mm,	Z = -243.572  mm,
	W = 0.000 deg,	P = 30.000 deg,	R = 138.564 deg
};
P[111]{
   GP1:
	UF : 0, UT : 1,		CONFIG : 'N U T, 0, 0, 0',
	X = 1121.406  mm,	Y = -194.769  mm,	Z = -243.735  mm,
	W = 0.000 deg,	P = 30.000 deg,	R = 138.564 deg
};
P[112]{
   GP1:
	UF : 0, UT : 1,		CONFIG : 'N U T, 0, 0, 0',
	X = 1122.516  mm,	Y = -192.540  mm,	Z = -243.921  mm,
	W = 0.000 deg,	P = 30.000 deg,	R = 138.564 deg
};
P[113]{
   GP1:
	UF : 0, UT : 1,		CONFIG : 'N U T, 0, 0, 0',
	X = 1123.866  mm,	Y = -190.347  mm,	Z = -244.186  mm,
	W = 0.000 deg,	P = 30.000 deg,	R = 138.564 deg
};
P[114]{
   GP1:
	UF : 0, UT : 1,		CONFIG : 'N U T, 0, 0, 0',
	X = 1125.391  mm,	Y = -188.183  mm,	Z = -244.520  mm,
	W = 0.000 deg,	P = 30.000 deg,	R = 138.564 deg
};
P[115]{
   GP1:
	UF : 0, UT : 1,		CONFIG : 'N U T, 0, 0, 0',
	X = 1127.116  mm,	Y = -186.071  mm,	Z = -244.949  mm,
	W = 0.000 deg,	P = 30.000 deg,	R = 138.564 deg
};
P[116]{
   GP1:
	UF : 0, UT : 1,		CONFIG : 'N U T, 0, 0, 0',
	X = 1128.852  mm,	Y = -184.055  mm,	Z = -245.422  mm,
	W = 0.000 deg,	P = 30.000 deg,	R = 138.564 deg
};
P[117]{
   GP1:
	UF : 0, UT : 1,		CONFIG : 'N U T, 0, 0, 0',
	X = 1130.567  mm,	Y = -182.020  mm,	Z = -245.891  mm,
	W = 0.000 deg,	P = 30.000 deg,	R = 138.564 deg
};
P[118]{
   GP1:
	UF : 0, UT : 1,		CONFIG : 'N U T, 0, 0, 0',
	X = 1136.827  mm,	Y = -184.064  mm,	Z = -246.437  mm,
	W = 0.000 deg,	P = 30.000 deg,	R = 138.564 deg
};
P[119]{
   GP1:
	UF : 0, UT : 1,		CONFIG : 'N U T, 0, 0, 0',
	X = 1138.756  mm,	Y = -182.098  mm,	Z = -247.064  mm,
	W = 0.000 deg,	P = 30.000 deg,	R = 138.564 deg
};
P[120]{
   GP1:
	UF : 0, UT : 1,		CONFIG : 'N U T, 0, 0, 0',
	X = 1140.692  mm,	Y = -180.114  mm,	Z = -247.691  mm,
	W = 0.000 deg,	P = 30.000 deg,	R = 138.564 deg
};
P[121]{
   GP1:
	UF : 0, UT : 1,		CONFIG : 'N U T, 0, 0, 0',
	X = 1142.706  mm,	Y = -178.120  mm,	Z = -248.323  mm,
	W = 0.000 deg,	P = 30.000 deg,	R = 138.564 deg
};
P[122]{
   GP1:
	UF : 0, UT : 1,		CONFIG : 'N U T, 0, 0, 0',
	X = 1144.679  mm,	Y = -176.124  mm,	Z = -248.923  mm,
	W = 0.000 deg,	P = 30.000 deg,	R = 138.564 deg
};
P[123]{
   GP1:
	UF : 0, UT : 1,		CONFIG : 'N U T, 0, 0, 0',
	X = 1146.672  mm,	Y = -174.164  mm,	Z = -249.521  mm,
	W = 0.000 deg,	P = 30.000 deg,	R = 143.780 deg
};
P[124]{
   GP1:
	UF : 0, UT : 1,		CONFIG : 'N U T, 0, 0, 0',
	X = 1148.812  mm,	Y = -172.154  mm,	Z = -250.145  mm,
	W = 0.000 deg,	P = 30.000 deg,	R = 155.588 deg
};
P[125]{
   GP1:
	UF : 0, UT : 1,		CONFIG : 'N U T, 0, 0, 0',
	X = 1150.873  mm,	Y = -170.091  mm,	Z = -250.729  mm,
	W = 0.000 deg,	P = 30.000 deg,	R = 166.990 deg
};
P[126]{
   GP1:
	UF : 0, UT : 1,		CONFIG : 'N U T, 0, 0, 0',
	X = 1152.823  mm,	Y = -168.028  mm,	Z = -251.274  mm,
	W = 0.000 deg,	P = 30.000 deg,	R = 178.073 deg
};
P[127]{
   GP1:
	UF : 0, UT : 1,		CONFIG : 'N U T, 0, 0, 0',
	X = 1154.702  mm,	Y = -165.912  mm,	Z = -251.786  mm,
	W = 0.000 deg,	P = 30.000 deg,	R = 178.073 deg
};
P[128]{
   GP1:
	UF : 0, UT : 1,		CONFIG : 'N U T, 0, 0, 0',
	X = 1156.373  mm,	Y = -163.727  mm,	Z = -252.214  mm,
	W = 0.000 deg,	P = 30.000 deg,	R = 178.073 deg
};
P[129]{
   GP1:
	UF : 0, UT : 1,		CONFIG : 'N U T, 0, 0, 0',
	X = 1157.798  mm,	Y = -161.510  mm,	Z = -252.559  mm,
	W = 0.000 deg,	P = 30.000 deg,	R = 178.073 deg
};
P[130]{
   GP1:
	UF : 0, UT : 1,		CONFIG : 'N U T, 0, 0, 0',
	X = 1158.984  mm,	Y = -159.238  mm,	Z = -252.834  mm,
	W = 0.000 deg,	P = 30.000 deg,	R = 178.073 deg
};
P[131]{
   GP1:
	UF : 0, UT : 1,		CONFIG : 'N U T, 0, 0, 0',
	X = 1159.871  mm,	Y = -156.926  mm,	Z = -253.028  mm,
	W = 0.000 deg,	P = 30.000 deg,	R = 178.073 deg
};
P[132]{
   GP1:
	UF : 0, UT : 1,		CONFIG : 'N U T, 0, 0, 0',
	X = 1160.489  mm,	Y = -154.603  mm,	Z = -253.150  mm,
	W = 0.000 deg,	P = 30.000 deg,	R = 178.073 deg
};
P[133]{
   GP1:
	UF : 0, UT : 1,		CONFIG : 'N U T, 0, 0, 0',
	X = 1160.820  mm,	Y = -152.331  mm,	Z = -253.205  mm,
	W = 0.000 deg,	P = 30.000 deg,	R = 178.073 deg
};
P[134]{
   GP1:
	UF : 0, UT : 1,		CONFIG : 'N U T, 0, 0, 0',
	X = 1160.988  mm,	Y = -150.188  mm,	Z = -253.214  mm,
	W = 0.000 deg,	P = 30.000 deg,	R = 178.073 deg
};
P[135]{
   GP1:
	UF : 0, UT : 1,		CONFIG : 'N U T, 0, 0, 0',
	X = 1161.088  mm,	Y = -148.114  mm,	Z = -253.219  mm,
	W = 0.000 deg,	P = 30.000 deg,	R = 178.073 deg
};
P[136]{
   GP1:
	UF : 0, UT : 1,		CONFIG : 'N U T, 0, 0, 0',
	X = 1155.146  mm,	Y = -145.938  mm,	Z = -253.222  mm,
	W = 0.000 deg,	P = 30.000 deg,	R = 178.073 deg
};
P[137]{
   GP1:
	UF : 0, UT : 1,		CONFIG : 'N U T, 0, 0, 0',
	X = 1155.172  mm,	Y = -143.961  mm,	Z = -253.221  mm,
	W = 0.000 deg,	P = 30.000 deg,	R = 178.073 deg
};
P[138]{
   GP1:
	UF : 0, UT : 1,		CONFIG : 'N U T, 0, 0, 0',
	X = 1155.197  mm,	Y = -141.970  mm,	Z = -253.217  mm,
	W = 0.000 deg,	P = 30.000 deg,	R = 178.073 deg
};
P[139]{
   GP1:
	UF : 0, UT : 1,		CONFIG : 'N U T, 0, 0, 0',
	X = 1155.212  mm,	Y = -139.985  mm,	Z = -253.211  mm,
	W = 0.000 deg,	P = 30.000 deg,	R = 178.073 deg
};
P[140]{
   GP1:
	UF : 0, UT : 1,		CONFIG : 'N U T, 0, 0, 0',
	X = 1155.217  mm,	Y = -137.995  mm,	Z = -253.205  mm,
	W = 0.000 deg,	P = 30.000 deg,	R = 178.073 deg
};
P[141]{
   GP1:
	UF : 0, UT : 1,		CONFIG : 'N U T, 0, 0, 0',
	X = 1155.219  mm,	Y = -135.999  mm,	Z = -253.193  mm,
	W = 0.000 deg,	P = 30.000 deg,	R = 178.073 deg
};
P[142]{
   GP1:
	UF : 0, UT : 1,		CONFIG : 'N U T, 0, 0, 0',
	X = 1155.218  mm,	Y = -134.001  mm,	Z = -253.170  mm,
	W = 0.000 deg,	P = 30.000 deg,	R = 178.073 deg
};
P[143]{
   GP1:
	UF : 0, UT : 1,		CONFIG : 'N U T, 0, 0, 0',
	X = 1155.217  mm,	Y = -132.002  mm,	Z = -253.139  mm,
	W = 0.000 deg,	P = 30.000 deg,	R = 178.073 deg
};
P[144]{
   GP1:
	UF : 0, UT : 1,		CONFIG : 'N U T, 0, 0, 0',
	X = 1155.216  mm,	Y = -130.009  mm,	Z = -253.105  mm,
	W = 0.000 deg,	P = 30.000 deg,	R = 178.073 deg
};
P[145]{
   GP1:
	UF : 0, UT : 1,		CONFIG : 'N U T, 0, 0, 0',
	X = 1155.205  mm,	Y = -128.023  mm,	Z = -253.067  mm,
	W = 0.000 deg,	P = 30.000 deg,	R = 178.073 deg
};
P[146]{
   GP1:
	UF : 0, UT : 1,		CONFIG : 'N U T, 0, 0, 0',
	X = 1155.186  mm,	Y = -126.036  mm,	Z = -253.027  mm,
	W = 0.000 deg,	P = 30.000 deg,	R = 178.073 deg
};
P[147]{
   GP1:
	UF : 0, UT : 1,		CONFIG : 'N U T, 0, 0, 0',
	X = 1155.158  mm,	Y = -124.052  mm,	Z = -252.981  mm,
	W = 0.000 deg,	P = 30.000 deg,	R = 178.073 deg
};
P[148]{
   GP1:
	UF : 0, UT : 1,		CONFIG : 'N U T, 0, 0, 0',
	X = 1155.117  mm,	Y = -122.072  mm,	Z = -252.936  mm,
	W = 0.000 deg,	P = 30.000 deg,	R = 178.073 deg
};
P[149]{
   GP1:
	UF : 0, UT : 1,		CONFIG : 'N U T, 0, 0, 0',
	X = 1155.064  mm,	Y = -120.097  mm,	Z = -252.893  mm,
	W = 0.000 deg,	P = 30.000 deg,	R = 178.073 deg
};
P[150]{
   GP1:
	UF : 0, UT : 1,		CONFIG : 'N U T, 0, 0, 0',
	X = 1154.989  mm,	Y = -118.119  mm,	Z = -252.846  mm,
	W = 0.000 deg,	P = 30.000 deg,	R = 178.073 deg
};
P[151]{
   GP1:
	UF : 0, UT : 1,		CONFIG : 'N U T, 0, 0, 0',
	X = 1154.906  mm,	Y = -116.141  mm,	Z = -252.802  mm,
	W = 0.000 deg,	P = 30.000 deg,	R = 178.073 deg
};
P[152]{
   GP1:
	UF : 0, UT : 1,		CONFIG : 'N U T, 0, 0, 0',
	X = 1154.805  mm,	Y = -114.187  mm,	Z = -252.752  mm,
	W = 0.000 deg,	P = 30.000 deg,	R = 178.073 deg
};
P[153]{
   GP1:
	UF : 0, UT : 1,		CONFIG : 'N U T, 0, 0, 0',
	X = 1154.660  mm,	Y = -112.210  mm,	Z = -252.687  mm,
	W = 0.000 deg,	P = 30.000 deg,	R = 178.073 deg
};
P[154]{
   GP1:
	UF : 0, UT : 1,		CONFIG : 'N U T, 0, 0, 0',
	X = 1154.530  mm,	Y = -110.261  mm,	Z = -252.627  mm,
	W = 0.000 deg,	P = 30.000 deg,	R = 178.073 deg
};
P[155]{
   GP1:
	UF : 0, UT : 1,		CONFIG : 'N U T, 0, 0, 0',
	X = 1154.323  mm,	Y = -108.348  mm,	Z = -252.540  mm,
	W = 0.000 deg,	P = 30.000 deg,	R = -173.463 deg
};
P[156]{
   GP1:
	UF : 0, UT : 1,		CONFIG : 'N U T, 0, 0, 0',
	X = 1160.020  mm,	Y = -105.565  mm,	Z = -252.445  mm,
	W = 0.000 deg,	P = 30.000 deg,	R = -163.857 deg
};
P[157]{
   GP1:
	UF : 0, UT : 1,		CONFIG : 'N U T, 0, 0, 0',
	X = 1159.659  mm,	Y = -103.413  mm,	Z = -252.323  mm,
	W = 0.000 deg,	P = 30.000 deg,	R = -154.185 deg
};
P[158]{
   GP1:
	UF : 0, UT : 1,		CONFIG : 'N U T, 0, 0, 0',
	X = 1159.143  mm,	Y = -101.195  mm,	Z = -252.166  mm,
	W = 0.000 deg,	P = 30.000 deg,	R = -144.384 deg
};
P[159]{
   GP1:
	UF : 0, UT : 1,		CONFIG : 'N U T, 0, 0, 0',
	X = 1158.378  mm,	Y = -98.860  mm,	Z = -251.954  mm,
	W = 0.000 deg,	P = 30.000 deg,	R = -134.321 deg
};
P[160]{
   GP1:
	UF : 0, UT : 1,		CONFIG : 'N U T, 0, 0, 0',
	X = 1157.140  mm,	Y = -96.388  mm,	Z = -251.642  mm,
	W = 0.000 deg,	P = 30.000 deg,	R = -134.321 deg
};
P[161]{
   GP1:
	UF : 0, UT : 1,		CONFIG : 'N U T, 0, 0, 0',
	X = 1155.428  mm,	Y = -94.165  mm,	Z = -251.155  mm,
	W = 0.000 deg,	P = 30.000 deg,	R = -134.321 deg
};
P[162]{
   GP1:
	UF : 0, UT : 1,		CONFIG : 'N U T, 0, 0, 0',
	X = 1153.784  mm,	Y = -92.034  mm,	Z = -250.672  mm,
	W = 0.000 deg,	P = 30.000 deg,	R = -134.321 deg
};
P[163]{
   GP1:
	UF : 0, UT : 1,		CONFIG : 'N U T, 0, 0, 0',
	X = 1151.697  mm,	Y = -89.872  mm,	Z = -250.050  mm,
	W = 0.000 deg,	P = 30.000 deg,	R = -134.321 deg
};
P[164]{
   GP1:
	UF : 0, UT : 1,		CONFIG : 'N U T, 0, 0, 0',
	X = 1145.417  mm,	Y = -92.166  mm,	Z = -249.386  mm,
	W = 0.000 deg,	P = 30.000 deg,	R = -134.321 deg
};
P[165]{
   GP1:
	UF : 0, UT : 1,		CONFIG : 'N U T, 0, 0, 0',
	X = 1143.404  mm,	Y = -90.232  mm,	Z = -248.716  mm,
	W = 0.000 deg,	P = 30.000 deg,	R = -134.321 deg
};
P[166]{
   GP1:
	UF : 0, UT : 1,		CONFIG : 'N U T, 0, 0, 0',
	X = 1141.045  mm,	Y = -88.243  mm,	Z = -247.951  mm,
	W = 0.000 deg,	P = 30.000 deg,	R = -134.321 deg
};
P[167]{
   GP1:
	UF : 0, UT : 1,		CONFIG : 'N U T, 0, 0, 0',
	X = 1143.006  mm,	Y = -81.861  mm,	Z = -247.247  mm,
	W = 0.000 deg,	P = 30.000 deg,	R = -134.321 deg
};
P[168]{
   GP1:
	UF : 0, UT : 1,		CONFIG : 'N U T, 0, 0, 0',
	X = 1136.950  mm,	Y = -84.220  mm,	Z = -246.589  mm,
	W = 0.000 deg,	P = 30.000 deg,	R = -134.321 deg
};
P[169]{
   GP1:
	UF : 0, UT : 1,		CONFIG : 'N U T, 0, 0, 0',
	X = 1134.585  mm,	Y = -82.307  mm,	Z = -245.775  mm,
	W = 0.000 deg,	P = 30.000 deg,	R = -134.321 deg
};
P[170]{
   GP1:
	UF : 0, UT : 1,		CONFIG : 'N U T, 0, 0, 0',
	X = 1132.203  mm,	Y = -80.277  mm,	Z = -245.068  mm,
	W = 0.000 deg,	P = 30.000 deg,	R = -134.321 deg
};
P[171]{
   GP1:
	UF : 0, UT : 1,		CONFIG : 'N U T, 0, 0, 0',
	X = 1129.899  mm,	Y = -78.289  mm,	Z = -244.382  mm,
	W = 0.000 deg,	P = 30.000 deg,	R = -139.413 deg
};
P[172]{
   GP1:
	UF : 0, UT : 1,		CONFIG : 'N U T, 0, 0, 0',
	X = 1127.418  mm,	Y = -76.221  mm,	Z = -243.695  mm,
	W = 0.000 deg,	P = 30.000 deg,	R = -154.318 deg
};
P[173]{
   GP1:
	UF : 0, UT : 1,		CONFIG : 'N U T, 0, 0, 0',
	X = 1125.296  mm,	Y = -74.105  mm,	Z = -243.172  mm,
	W = 0.000 deg,	P = 30.000 deg,	R = -167.715 deg
};
P[174]{
   GP1:
	UF : 0, UT : 1,		CONFIG : 'N U T, 0, 0, 0',
	X = 1123.249  mm,	Y = -71.989  mm,	Z = -242.684  mm,
	W = 0.000 deg,	P = 30.000 deg,	R = 179.119 deg
};
P[175]{
   GP1:
	UF : 0, UT : 1,		CONFIG : 'N U T, 0, 0, 0',
	X = 1121.381  mm,	Y = -69.644  mm,	Z = -242.323  mm,
	W = 0.000 deg,	P = 30.000 deg,	R = 179.119 deg
};
P[176]{
   GP1:
	UF : 0, UT : 1,		CONFIG : 'N U T, 0, 0, 0',
	X = 1120.115  mm,	Y = -67.176  mm,	Z = -242.141  mm,
	W = 0.000 deg,	P = 30.000 deg,	R = 179.119 deg
};
P[177]{
   GP1:
	UF : 0, UT : 1,		CONFIG : 'N U T, 0, 0, 0',
	X = 1119.303  mm,	Y = -64.830  mm,	Z = -242.009  mm,
	W = 0.000 deg,	P = 30.000 deg,	R = 179.119 deg
};
P[178]{
   GP1:
	UF : 0, UT : 1,		CONFIG : 'N U T, 0, 0, 0',
	X = 1118.769  mm,	Y = -62.522  mm,	Z = -241.934  mm,
	W = 0.000 deg,	P = 30.000 deg,	R = 179.119 deg
};
P[179]{
   GP1:
	UF : 0, UT : 1,		CONFIG : 'N U T, 0, 0, 0',
	X = 1118.494  mm,	Y = -60.294  mm,	Z = -241.902  mm,
	W = 0.000 deg,	P = 30.000 deg,	R = 179.119 deg
};
P[180]{
   GP1:
	UF : 0, UT : 1,		CONFIG : 'N U T, 0, 0, 0',
	X = 1118.333  mm,	Y = -58.157  mm,	Z = -241.866  mm,
	W = 0.000 deg,	P = 30.000 deg,	R = 179.119 deg
};
P[181]{
   GP1:
	UF : 0, UT : 1,		CONFIG : 'N U T, 0, 0, 0',
	X = 1118.270  mm,	Y = -56.067  mm,	Z = -241.849  mm,
	W = 0.000 deg,	P = 30.000 deg,	R = 179.119 deg
};
P[182]{
   GP1:
	UF : 0, UT : 1,		CONFIG : 'N U T, 0, 0, 0',
	X = 1118.239  mm,	Y = -54.032  mm,	Z = -241.832  mm,
	W = 0.000 deg,	P = 30.000 deg,	R = 179.119 deg
};
P[183]{
   GP1:
	UF : 0, UT : 1,		CONFIG : 'N U T, 0, 0, 0',
	X = 1118.227  mm,	Y = -52.014  mm,	Z = -241.817  mm,
	W = 0.000 deg,	P = 30.000 deg,	R = 179.119 deg
};
P[184]{
   GP1:
	UF : 0, UT : 1,		CONFIG : 'N U T, 0, 0, 0',
	X = 1118.220  mm,	Y = -50.006  mm,	Z = -241.801  mm,
	W = 0.000 deg,	P = 30.000 deg,	R = 179.119 deg
};
P[185]{
   GP1:
	UF : 0, UT : 1,		CONFIG : 'N U T, 0, 0, 0',
	X = 1118.218  mm,	Y = -48.001  mm,	Z = -241.788  mm,
	W = 0.000 deg,	P = 30.000 deg,	R = 179.119 deg
};
P[186]{
   GP1:
	UF : 0, UT : 1,		CONFIG : 'N U T, 0, 0, 0',
	X = 1118.218  mm,	Y = -45.997  mm,	Z = -241.781  mm,
	W = 0.000 deg,	P = 30.000 deg,	R = 179.119 deg
};
P[187]{
   GP1:
	UF : 0, UT : 1,		CONFIG : 'N U T, 0, 0, 0',
	X = 1118.222  mm,	Y = -43.991  mm,	Z = -241.778  mm,
	W = 0.000 deg,	P = 30.000 deg,	R = 179.119 deg
};
P[188]{
   GP1:
	UF : 0, UT : 1,		CONFIG : 'N U T, 0, 0, 0',
	X = 1118.231  mm,	Y = -41.986  mm,	Z = -241.773  mm,
	W = 0.000 deg,	P = 30.000 deg,	R = 179.119 deg
};
P[189]{
   GP1:
	UF : 0, UT : 1,		CONFIG : 'N U T, 0, 0, 0',
	X = 1118.241  mm,	Y = -39.981  mm,	Z = -241.773  mm,
	W = 0.000 deg,	P = 30.000 deg,	R = 179.119 deg
};
P[190]{
   GP1:
	UF : 0, UT : 1,		CONFIG : 'N U T, 0, 0, 0',
	X = 1118.257  mm,	Y = -37.966  mm,	Z = -241.772  mm,
	W = 0.000 deg,	P = 30.000 deg,	R = 179.119 deg
};
P[191]{
   GP1:
	UF : 0, UT : 1,		CONFIG : 'N U T, 0, 0, 0',
	X = 1124.285  mm,	Y = -36.050  mm,	Z = -241.773  mm,
	W = 0.000 deg,	P = 30.000 deg,	R = 179.119 deg
};
P[192]{
   GP1:
	UF : 0, UT : 1,		CONFIG : 'N U T, 0, 0, 0',
	X = 1124.322  mm,	Y = -34.062  mm,	Z = -241.770  mm,
	W = 0.000 deg,	P = 30.000 deg,	R = 179.119 deg
};
P[193]{
   GP1:
	UF : 0, UT : 1,		CONFIG : 'N U T, 0, 0, 0',
	X = 1124.367  mm,	Y = -32.076  mm,	Z = -241.755  mm,
	W = 0.000 deg,	P = 30.000 deg,	R = 179.119 deg
};
P[194]{
   GP1:
	UF : 0, UT : 1,		CONFIG : 'N U T, 0, 0, 0',
	X = 1124.423  mm,	Y = -30.086  mm,	Z = -241.738  mm,
	W = 0.000 deg,	P = 30.000 deg,	R = 179.119 deg
};
P[195]{
   GP1:
	UF : 0, UT : 1,		CONFIG : 'N U T, 0, 0, 0',
	X = 1124.481  mm,	Y = -28.096  mm,	Z = -241.725  mm,
	W = 0.000 deg,	P = 30.000 deg,	R = 179.119 deg
};
P[196]{
   GP1:
	UF : 0, UT : 1,		CONFIG : 'N U T, 0, 0, 0',
	X = 1124.551  mm,	Y = -26.108  mm,	Z = -241.715  mm,
	W = 0.000 deg,	P = 30.000 deg,	R = 179.119 deg
};
P[197]{
   GP1:
	UF : 0, UT : 1,		CONFIG : 'N U T, 0, 0, 0',
	X = 1124.625  mm,	Y = -24.113  mm,	Z = -241.702  mm,
	W = 0.000 deg,	P = 30.000 deg,	R = 179.119 deg
};
P[198]{
   GP1:
	UF : 0, UT : 1,		CONFIG : 'N U T, 0, 0, 0',
	X = 1124.700  mm,	Y = -22.143  mm,	Z = -241.688  mm,
	W = 0.000 deg,	P = 30.000 deg,	R = 179.119 deg
};
P[199]{
   GP1:
	UF : 0, UT : 1,		CONFIG : 'N U T, 0, 0, 0',
	X = 1124.811  mm,	Y = -20.198  mm,	Z = -241.674  mm,
	W = 0.000 deg,	P = 30.000 deg,	R = 179.119 deg
};
P[200]{
   GP1:
	UF : 0, UT : 1,		CONFIG : 'N U T, 0, 0, 0',
	X = 1124.956  mm,	Y = -18.273  mm,	Z = -241.672  mm,
	W = 0.000 deg,	P = 30.000 deg,	R = 179.119 deg
};
P[201]{
   GP1:
	UF : 0, UT : 1,		CONFIG : 'N U T, 0, 0, 0',
	X = 1119.209  mm,	Y = -15.610  mm,	Z = -241.677  mm,
	W = 0.000 deg,	P = 30.000 deg,	R = 171.666 deg
};
P[202]{
   GP1:
	UF : 0, UT : 1,		CONFIG : 'N U T, 0, 0, 0',
	X = 1119.533  mm,	Y = -13.513  mm,	Z = -241.682  mm,
	W = 0.000 deg,	P = 30.000 deg,	R = 163.164 deg
};
P[203]{
   GP1:
	UF : 0, UT : 1,		CONFIG : 'N U T, 0, 0, 0',
	X = 1119.900  mm,	Y = -11.407  mm,	Z = -241.690  mm,
	W = 0.000 deg,	P = 30.000 deg,	R = 154.635 deg
};
P[204]{
   GP1:
	UF : 0, UT : 1,		CONFIG : 'N U T, 0, 0, 0',
	X = 1120.417  mm,	Y = -9.167  mm,	Z = -241.712  mm,
	W = 0.000 deg,	P = 30.000 deg,	R = 146.015 deg
};
P[205]{
   GP1:
	UF : 0, UT : 1,		CONFIG : 'N U T, 0, 0, 0',
	X = 1121.198  mm,	Y = -6.919  mm,	Z = -241.799  mm,
	W = 0.000 deg,	P = 30.000 deg,	R = 137.109 deg
};
P[206]{
   GP1:
	UF : 0, UT : 1,		CONFIG : 'N U T, 0, 0, 0',
	X = 1122.128  mm,	Y = -4.725  mm,	Z = -241.944  mm,
	W = 0.000 deg,	P = 30.000 deg,	R = 137.109 deg
};
P[207]{
   GP1:
	UF : 0, UT : 1,		CONFIG : 'N U T, 0, 0, 0',
	X = 1123.268  mm,	Y = -2.514  mm,	Z = -242.119  mm,
	W = 0.000 deg,	P = 30.000 deg,	R = 137.109 deg
};
P[208]{
   GP1:
	UF : 0, UT : 1,		CONFIG : 'N U T, 0, 0, 0',
	X = 1124.638  mm,	Y = -0.322  mm,	Z = -242.327  mm,
	W = 0.000 deg,	P = 30.000 deg,	R = 137.109 deg
};
P[209]{
   GP1:
	UF : 0, UT : 1,		CONFIG : 'N U T, 0, 0, 0',
	X = 1126.198  mm,	Y = 1.832  mm,	Z = -242.635  mm,
	W = 0.000 deg,	P = 30.000 deg,	R = 137.109 deg
};
P[210]{
   GP1:
	UF : 0, UT : 1,		CONFIG : 'N U T, 0, 0, 0',
	X = 1127.926  mm,	Y = 3.946  mm,	Z = -243.021  mm,
	W = 0.000 deg,	P = 30.000 deg,	R = 137.109 deg
};
P[211]{
   GP1:
	UF : 0, UT : 1,		CONFIG : 'N U T, 0, 0, 0',
	X = 1129.775  mm,	Y = 6.030  mm,	Z = -243.485  mm,
	W = 0.000 deg,	P = 30.000 deg,	R = 137.109 deg
};
P[212]{
   GP1:
	UF : 0, UT : 1,		CONFIG : 'N U T, 0, 0, 0',
	X = 1136.030  mm,	Y = 3.904  mm,	Z = -244.017  mm,
	W = 0.000 deg,	P = 30.000 deg,	R = 137.109 deg
};
P[213]{
   GP1:
	UF : 0, UT : 1,		CONFIG : 'N U T, 0, 0, 0',
	X = 1137.990  mm,	Y = 5.857  mm,	Z = -244.583  mm,
	W = 0.000 deg,	P = 30.000 deg,	R = 137.109 deg
};
P[214]{
   GP1:
	UF : 0, UT : 1,		CONFIG : 'N U T, 0, 0, 0',
	X = 1140.036  mm,	Y = 7.829  mm,	Z = -245.211  mm,
	W = 0.000 deg,	P = 30.000 deg,	R = 137.109 deg
};
P[215]{
   GP1:
	UF : 0, UT : 1,		CONFIG : 'N U T, 0, 0, 0',
	X = 1142.119  mm,	Y = 9.796  mm,	Z = -245.909  mm,
	W = 0.000 deg,	P = 30.000 deg,	R = 137.109 deg
};
P[216]{
   GP1:
	UF : 0, UT : 1,		CONFIG : 'N U T, 0, 0, 0',
	X = 1144.300  mm,	Y = 11.766  mm,	Z = -246.627  mm,
	W = 0.000 deg,	P = 30.000 deg,	R = 137.109 deg
};
P[217]{
   GP1:
	UF : 0, UT : 1,		CONFIG : 'N U T, 0, 0, 0',
	X = 1146.552  mm,	Y = 13.770  mm,	Z = -247.337  mm,
	W = 0.000 deg,	P = 30.000 deg,	R = 141.576 deg
};
P[218]{
   GP1:
	UF : 0, UT : 1,		CONFIG : 'N U T, 0, 0, 0',
	X = 1148.812  mm,	Y = 15.829  mm,	Z = -248.018  mm,
	W = 0.000 deg,	P = 30.000 deg,	R = 153.597 deg
};
P[219]{
   GP1:
	UF : 0, UT : 1,		CONFIG : 'N U T, 0, 0, 0',
	X = 1150.848  mm,	Y = 17.866  mm,	Z = -248.621  mm,
	W = 0.000 deg,	P = 30.000 deg,	R = 164.994 deg
};
P[220]{
   GP1:
	UF : 0, UT : 1,		CONFIG : 'N U T, 0, 0, 0',
	X = 1152.917  mm,	Y = 19.886  mm,	Z = -249.239  mm,
	W = 0.000 deg,	P = 30.000 deg,	R = 176.549 deg
};
P[221]{
   GP1:
	UF : 0, UT : 1,		CONFIG : 'N U T, 0, 0, 0',
	X = 1154.930  mm,	Y = 21.979  mm,	Z = -249.811  mm,
	W = 0.000 deg,	P = 30.000 deg,	R = 176.549 deg
};
P[222]{
   GP1:
	UF : 0, UT : 1,		CONFIG : 'N U T, 0, 0, 0',
	X = 1156.800  mm,	Y = 24.157  mm,	Z = -250.312  mm,
	W = 0.000 deg,	P = 30.000 deg,	R = 176.549 deg
};
P[223]{
   GP1:
	UF : 0, UT : 1,		CONFIG : 'N U T, 0, 0, 0',
	X = 1158.362  mm,	Y = 26.396  mm,	Z = -250.707  mm,
	W = 0.000 deg,	P = 30.000 deg,	R = 176.549 deg
};
P[224]{
   GP1:
	UF : 0, UT : 1,		CONFIG : 'N U T, 0, 0, 0',
	X = 1159.628  mm,	Y = 28.621  mm,	Z = -251.031  mm,
	W = 0.000 deg,	P = 30.000 deg,	R = 176.549 deg
};
P[225]{
   GP1:
	UF : 0, UT : 1,		CONFIG : 'N U T, 0, 0, 0',
	X = 1160.661  mm,	Y = 30.835  mm,	Z = -251.293  mm,
	W = 0.000 deg,	P = 30.000 deg,	R = 176.549 deg
};
P[226]{
   GP1:
	UF : 0, UT : 1,		CONFIG : 'N U T, 0, 0, 0',
	X = 1161.532  mm,	Y = 33.167  mm,	Z = -251.506  mm,
	W = 0.000 deg,	P = 30.000 deg,	R = 176.549 deg
};
P[227]{
   GP1:
	UF : 0, UT : 1,		CONFIG : 'N U T, 0, 0, 0',
	X = 1162.016  mm,	Y = 35.531  mm,	Z = -251.612  mm,
	W = 0.000 deg,	P = 30.000 deg,	R = 176.549 deg
};
P[228]{
   GP1:
	UF : 0, UT : 1,		CONFIG : 'N U T, 0, 0, 0',
	X = 1162.273  mm,	Y = 37.748  mm,	Z = -251.670  mm,
	W = 0.000 deg,	P = 30.000 deg,	R = 176.549 deg
};
P[229]{
   GP1:
	UF : 0, UT : 1,		CONFIG : 'N U T, 0, 0, 0',
	X = 1156.393  mm,	Y = 40.113  mm,	Z = -251.686  mm,
	W = 0.000 deg,	P = 30.000 deg,	R = 176.549 deg
};
P[230]{
   GP1:
	UF : 0, UT : 1,		CONFIG : 'N U T, 0, 0, 0',
	X = 1156.435  mm,	Y = 42.057  mm,	Z = -251.683  mm,
	W = 0.000 deg,	P = 30.000 deg,	R = 176.549 deg
};
P[231]{
   GP1:
	UF : 0, UT : 1,		CONFIG : 'N U T, 0, 0, 0',
	X = 1156.467  mm,	Y = 44.045  mm,	Z = -251.674  mm,
	W = 0.000 deg,	P = 30.000 deg,	R = 176.549 deg
};
P[232]{
   GP1:
	UF : 0, UT : 1,		CONFIG : 'N U T, 0, 0, 0',
	X = 1156.495  mm,	Y = 46.040  mm,	Z = -251.658  mm,
	W = 0.000 deg,	P = 30.000 deg,	R = 176.549 deg
};
P[233]{
   GP1:
	UF : 0, UT : 1,		CONFIG : 'N U T, 0, 0, 0',
	X = 1156.520  mm,	Y = 48.036  mm,	Z = -251.636  mm,
	W = 0.000 deg,	P = 30.000 deg,	R = 176.549 deg
};
P[234]{
   GP1:
	UF : 0, UT : 1,		CONFIG : 'N U T, 0, 0, 0',
	X = 1156.543  mm,	Y = 50.032  mm,	Z = -251.615  mm,
	W = 0.000 deg,	P = 30.000 deg,	R = 176.549 deg
};
P[235]{
   GP1:
	UF : 0, UT : 1,		CONFIG : 'N U T, 0, 0, 0',
	X = 1156.563  mm,	Y = 52.022  mm,	Z = -251.590  mm,
	W = 0.000 deg,	P = 30.000 deg,	R = 176.549 deg
};
P[236]{
   GP1:
	UF : 0, UT : 1,		CONFIG : 'N U T, 0, 0, 0',
	X = 1156.572  mm,	Y = 54.006  mm,	Z = -251.564  mm,
	W = 0.000 deg,	P = 30.000 deg,	R = 176.549 deg
};
P[237]{
   GP1:
	UF : 0, UT : 1,		CONFIG : 'N U T, 0, 0, 0',
	X = 1156.570  mm,	Y = 55.993  mm,	Z = -251.540  mm,
	W = 0.000 deg,	P = 30.000 deg,	R = 176.549 deg
};
P[238]{
   GP1:
	UF : 0, UT : 1,		CONFIG : 'N U T, 0, 0, 0',
	X = 1156.562  mm,	Y = 57.984  mm,	Z = -251.513  mm,
	W = 0.000 deg,	P = 30.000 deg,	R = 176.549 deg
};
P[239]{
   GP1:
	UF : 0, UT : 1,		CONFIG : 'N U T, 0, 0, 0',
	X = 1156.549  mm,	Y = 59.975  mm,	Z = -251.489  mm,
	W = 0.000 deg,	P = 30.000 deg,	R = 176.549 deg
};
P[240]{
   GP1:
	UF : 0, UT : 1,		CONFIG : 'N U T, 0, 0, 0',
	X = 1156.529  mm,	Y = 61.960  mm,	Z = -251.463  mm,
	W = 0.000 deg,	P = 30.000 deg,	R = 176.549 deg
};
P[241]{
   GP1:
	UF : 0, UT : 1,		CONFIG : 'N U T, 0, 0, 0',
	X = 1156.496  mm,	Y = 63.946  mm,	Z = -251.431  mm,
	W = 0.000 deg,	P = 30.000 deg,	R = 176.549 deg
};
P[242]{
   GP1:
	UF : 0, UT : 1,		CONFIG : 'N U T, 0, 0, 0',
	X = 1156.457  mm,	Y = 65.940  mm,	Z = -251.396  mm,
	W = 0.000 deg,	P = 30.000 deg,	R = 176.549 deg
};
P[243]{
   GP1:
	UF : 0, UT : 1,		CONFIG : 'N U T, 0, 0, 0',
	X = 1156.417  mm,	Y = 67.931  mm,	Z = -251.362  mm,
	W = 0.000 deg,	P = 30.000 deg,	R = 176.549 deg
};
P[244]{
   GP1:
	UF : 0, UT : 1,		CONFIG : 'N U T, 0, 0, 0',
	X = 1156.365  mm,	Y = 69.911  mm,	Z = -251.325  mm,
	W = 0.000 deg,	P = 30.000 deg,	R = 176.549 deg
};
P[245]{
   GP1:
	UF : 0, UT : 1,		CONFIG : 'N U T, 0, 0, 0',
	X = 1156.299  mm,	Y = 71.890  mm,	Z = -251.285  mm,
	W = 0.000 deg,	P = 30.000 deg,	R = 176.549 deg
};
P[246]{
   GP1:
	UF : 0, UT : 1,		CONFIG : 'N U T, 0, 0, 0',
	X = 1156.219  mm,	Y = 73.886  mm,	Z = -251.240  mm,
	W = 0.000 deg,	P = 30.000 deg,	R = 176.549 deg
};
P[247]{
   GP1:
	UF : 0, UT : 1,		CONFIG : 'N U T, 0, 0, 0',
	X = 1156.147  mm,	Y = 75.888  mm,	Z = -251.200  mm,
	W = 0.000 deg,	P = 30.000 deg,	R = 176.549 deg
};
P[248]{
   GP1:
	UF : 0, UT : 1,		CONFIG : 'N U T, 0, 0, 0',
	X = 1156.071  mm,	Y = 77.869  mm,	Z = -251.160  mm,
	W = 0.000 deg,	P = 30.000 deg,	R = 176.549 deg
};
P[249]{
   GP1:
	UF : 0, UT : 1,		CONFIG : 'N U T, 0, 0, 0',
	X = 1161.963  mm,	Y = 80.203  mm,	Z = -251.114  mm,
	W = 0.000 deg,	P = 30.000 deg,	R = -174.774 deg
};
P[250]{
   GP1:
	UF : 0, UT : 1,		CONFIG : 'N U T, 0, 0, 0',
	X = 1161.779  mm,	Y = 82.326  mm,	Z = -251.043  mm,
	W = 0.000 deg,	P = 30.000 deg,	R = -165.306 deg
};
P[251]{
   GP1:
	UF : 0, UT : 1,		CONFIG : 'N U T, 0, 0, 0',
	X = 1161.493  mm,	Y = 84.484  mm,	Z = -250.944  mm,
	W = 0.000 deg,	P = 30.000 deg,	R = -155.786 deg
};
P[252]{
   GP1:
	UF : 0, UT : 1,		CONFIG : 'N U T, 0, 0, 0',
	X = 1161.060  mm,	Y = 86.701  mm,	Z = -250.812  mm,
	W = 0.000 deg,	P = 30.000 deg,	R = -146.162 deg
};
P[253]{
   GP1:
	UF : 0, UT : 1,		CONFIG : 'N U T, 0, 0, 0',
	X = 1160.391  mm,	Y = 89.022  mm,	Z = -250.623  mm,
	W = 0.000 deg,	P = 30.000 deg,	R = -136.316 deg
};
P[254]{
   GP1:
	UF : 0, UT : 1,		CONFIG : 'N U T, 0, 0, 0',
	X = 1159.393  mm,	Y = 91.308  mm,	Z = -250.332  mm,
	W = 0.000 deg,	P = 30.000 deg,	R = -136.316 deg
};
P[255]{
   GP1:
	UF : 0, UT : 1,		CONFIG : 'N U T, 0, 0, 0',
	X = 1158.166  mm,	Y = 93.606  mm,	Z = -249.989  mm,
	W = 0.000 deg,	P = 30.000 deg,	R = -136.316 deg
};
P[256]{
   GP1:
	UF : 0, UT : 1,		CONFIG : 'N U T, 0, 0, 0',
	X = 1156.448  mm,	Y = 95.938  mm,	Z = -249.520  mm,
	W = 0.000 deg,	P = 30.000 deg,	R = -136.316 deg
};
P[257]{
   GP1:
	UF : 0, UT : 1,		CONFIG : 'N U T, 0, 0, 0',
	X = 1150.118  mm,	Y = 93.885  mm,	Z = -248.890  mm,
	W = 0.000 deg,	P = 30.000 deg,	R = -136.316 deg
};
P[258]{
   GP1:
	UF : 0, UT : 1,		CONFIG : 'N U T, 0, 0, 0',
	X = 1148.079  mm,	Y = 95.861  mm,	Z = -248.208  mm,
	W = 0.000 deg,	P = 30.000 deg,	R = -136.316 deg
};
P[259]{
   GP1:
	UF : 0, UT : 1,		CONFIG : 'N U T, 0, 0, 0',
	X = 1146.148  mm,	Y = 97.792  mm,	Z = -247.544  mm,
	W = 0.000 deg,	P = 30.000 deg,	R = -136.316 deg
};
P[260]{
   GP1:
	UF : 0, UT : 1,		CONFIG : 'N U T, 0, 0, 0',
	X = 1143.812  mm,	Y = 99.784  mm,	Z = -246.760  mm,
	W = 0.000 deg,	P = 30.000 deg,	R = -136.316 deg
};
P[261]{
   GP1:
	UF : 0, UT : 1,		CONFIG : 'N U T, 0, 0, 0',
	X = 1141.755  mm,	Y = 101.801  mm,	Z = -246.080  mm,
	W = 0.000 deg,	P = 30.000 deg,	R = -136.316 deg
};
P[262]{
   GP1:
	UF : 0, UT : 1,		CONFIG : 'N U T, 0, 0, 0',
	X = 1139.497  mm,	Y = 103.788  mm,	Z = -245.295  mm,
	W = 0.000 deg,	P = 30.000 deg,	R = -136.316 deg
};
P[263]{
   GP1:
	UF : 0, UT : 1,		CONFIG : 'N U T, 0, 0, 0',
	X = 1137.379  mm,	Y = 105.810  mm,	Z = -244.553  mm,
	W = 0.000 deg,	P = 30.000 deg,	R = -136.316 deg
};
P[264]{
   GP1:
	UF : 0, UT : 1,		CONFIG : 'N U T, 0, 0, 0',
	X = 1135.259  mm,	Y = 107.759  mm,	Z = -243.883  mm,
	W = 0.000 deg,	P = 30.000 deg,	R = -136.316 deg
};
P[265]{
   GP1:
	UF : 0, UT : 1,		CONFIG : 'N U T, 0, 0, 0',
	X = 1132.991  mm,	Y = 109.715  mm,	Z = -243.212  mm,
	W = 0.000 deg,	P = 30.000 deg,	R = -136.316 deg
};
P[266]{
   GP1:
	UF : 0, UT : 1,		CONFIG : 'N U T, 0, 0, 0',
	X = 1130.544  mm,	Y = 111.773  mm,	Z = -242.530  mm,
	W = 0.000 deg,	P = 30.000 deg,	R = -136.316 deg
};
P[267]{
   GP1:
	UF : 0, UT : 1,		CONFIG : 'N U T, 0, 0, 0',
	X = 1128.434  mm,	Y = 113.828  mm,	Z = -241.997  mm,
	W = 0.000 deg,	P = 30.000 deg,	R = -144.703 deg
};
P[268]{
   GP1:
	UF : 0, UT : 1,		CONFIG : 'N U T, 0, 0, 0',
	X = 1126.201  mm,	Y = 115.911  mm,	Z = -241.451  mm,
	W = 0.000 deg,	P = 30.000 deg,	R = -158.397 deg
};
P[269]{
   GP1:
	UF : 0, UT : 1,		CONFIG : 'N U T, 0, 0, 0',
	X = 1124.286  mm,	Y = 118.118  mm,	Z = -241.067  mm,
	W = 0.000 deg,	P = 30.000 deg,	R = -170.661 deg
};
P[270]{
   GP1:
	UF : 0, UT : 1,		CONFIG : 'N U T, 0, 0, 0',
	X = 1122.559  mm,	Y = 120.456  mm,	Z = -240.769  mm,
	W = 0.000 deg,	P = 30.000 deg,	R = 177.816 deg
};
P[271]{
   GP1:
	UF : 0, UT : 1,		CONFIG : 'N U T, 0, 0, 0',
	X = 1121.395  mm,	Y = 122.992  mm,	Z = -240.587  mm,
	W = 0.000 deg,	P = 30.000 deg,	R = 177.816 deg
};
P[272]{
   GP1:
	UF : 0, UT : 1,		CONFIG : 'N U T, 0, 0, 0',
	X = 1120.776  mm,	Y = 125.346  mm,	Z = -240.478  mm,
	W = 0.000 deg,	P = 30.000 deg,	R = 177.816 deg
};
P[273]{
   GP1:
	UF : 0, UT : 1,		CONFIG : 'N U T, 0, 0, 0',
	X = 1120.355  mm,	Y = 127.591  mm,	Z = -240.406  mm,
	W = 0.000 deg,	P = 30.000 deg,	R = 177.816 deg
};
P[274]{
   GP1:
	UF : 0, UT : 1,		CONFIG : 'N U T, 0, 0, 0',
	X = 1120.160  mm,	Y = 129.813  mm,	Z = -240.359  mm,
	W = 0.000 deg,	P = 30.000 deg,	R = 177.816 deg
};
P[275]{
   GP1:
	UF : 0, UT : 1,		CONFIG : 'N U T, 0, 0, 0',
	X = 1120.080  mm,	Y = 131.895  mm,	Z = -240.319  mm,
	W = 0.000 deg,	P = 30.000 deg,	R = 177.816 deg
};
P[276]{
   GP1:
	UF : 0, UT : 1,		CONFIG : 'N U T, 0, 0, 0',
	X = 1120.016  mm,	Y = 133.922  mm,	Z = -240.269  mm,
	W = 0.000 deg,	P = 30.000 deg,	R = 177.816 deg
};
P[277]{
   GP1:
	UF : 0, UT : 1,		CONFIG : 'N U T, 0, 0, 0',
	X = 1119.974  mm,	Y = 135.951  mm,	Z = -240.224  mm,
	W = 0.000 deg,	P = 30.000 deg,	R = 177.816 deg
};
P[278]{
   GP1:
	UF : 0, UT : 1,		CONFIG : 'N U T, 0, 0, 0',
	X = 1119.950  mm,	Y = 137.969  mm,	Z = -240.182  mm,
	W = 0.000 deg,	P = 30.000 deg,	R = 177.816 deg
};
P[279]{
   GP1:
	UF : 0, UT : 1,		CONFIG : 'N U T, 0, 0, 0',
	X = 1119.932  mm,	Y = 139.978  mm,	Z = -240.146  mm,
	W = 0.000 deg,	P = 30.000 deg,	R = 177.816 deg
};
P[280]{
   GP1:
	UF : 0, UT : 1,		CONFIG : 'N U T, 0, 0, 0',
	X = 1119.921  mm,	Y = 141.989  mm,	Z = -240.111  mm,
	W = 0.000 deg,	P = 30.000 deg,	R = 177.816 deg
};
P[281]{
   GP1:
	UF : 0, UT : 1,		CONFIG : 'N U T, 0, 0, 0',
	X = 1119.917  mm,	Y = 143.998  mm,	Z = -240.079  mm,
	W = 0.000 deg,	P = 30.000 deg,	R = 177.816 deg
};
P[282]{
   GP1:
	UF : 0, UT : 1,		CONFIG : 'N U T, 0, 0, 0',
	X = 1119.918  mm,	Y = 146.017  mm,	Z = -240.053  mm,
	W = 0.000 deg,	P = 30.000 deg,	R = 177.816 deg
};
P[283]{
   GP1:
	UF : 0, UT : 1,		CONFIG : 'N U T, 0, 0, 0',
	X = 1119.940  mm,	Y = 148.039  mm,	Z = -240.038  mm,
	W = 0.000 deg,	P = 30.000 deg,	R = 177.816 deg
};
P[284]{
   GP1:
	UF : 0, UT : 1,		CONFIG : 'N U T, 0, 0, 0',
	X = 1119.971  mm,	Y = 150.051  mm,	Z = -240.026  mm,
	W = 0.000 deg,	P = 30.000 deg,	R = 177.816 deg
};
P[285]{
   GP1:
	UF : 0, UT : 1,		CONFIG : 'N U T, 0, 0, 0',
	X = 1120.008  mm,	Y = 152.063  mm,	Z = -240.011  mm,
	W = 0.000 deg,	P = 30.000 deg,	R = 177.816 deg
};
P[286]{
   GP1:
	UF : 0, UT : 1,		CONFIG : 'N U T, 0, 0, 0',
	X = 1120.056  mm,	Y = 154.075  mm,	Z = -239.999  mm,
	W = 0.000 deg,	P = 30.000 deg,	R = 177.816 deg
};
P[287]{
   GP1:
	UF : 0, UT : 1,		CONFIG : 'N U T, 0, 0, 0',
	X = 1120.109  mm,	Y = 156.089  mm,	Z = -239.991  mm,
	W = 0.000 deg,	P = 30.000 deg,	R = 177.816 deg
};
P[288]{
   GP1:
	UF : 0, UT : 1,		CONFIG : 'N U T, 0, 0, 0',
	X = 1120.175  mm,	Y = 158.107  mm,	Z = -239.991  mm,
	W = 0.000 deg,	P = 30.000 deg,	R = 177.816 deg
};
P[289]{
   GP1:
	UF : 0, UT : 1,		CONFIG : 'N U T, 0, 0, 0',
	X = 1126.249  mm,	Y = 159.885  mm,	Z = -239.991  mm,
	W = 0.000 deg,	P = 30.000 deg,	R = 177.816 deg
};
P[290]{
   GP1:
	UF : 0, UT : 1,		CONFIG : 'N U T, 0, 0, 0',
	X = 1126.324  mm,	Y = 161.870  mm,	Z = -239.990  mm,
	W = 0.000 deg,	P = 30.000 deg,	R = 177.816 deg
};
P[291]{
   GP1:
	UF : 0, UT : 1,		CONFIG : 'N U T, 0, 0, 0',
	X = 1126.421  mm,	Y = 163.843  mm,	Z = -239.995  mm,
	W = 0.000 deg,	P = 30.000 deg,	R = 177.816 deg
};
P[292]{
   GP1:
	UF : 0, UT : 1,		CONFIG : 'N U T, 0, 0, 0',
	X = 1126.530  mm,	Y = 165.814  mm,	Z = -240.005  mm,
	W = 0.000 deg,	P = 30.000 deg,	R = 177.816 deg
};
P[293]{
   GP1:
	UF : 0, UT : 1,		CONFIG : 'N U T, 0, 0, 0',
	X = 1126.665  mm,	Y = 167.765  mm,	Z = -240.015  mm,
	W = 0.000 deg,	P = 30.000 deg,	R = 177.816 deg
};
P[294]{
   GP1:
	UF : 0, UT : 1,		CONFIG : 'N U T, 0, 0, 0',
	X = 1126.836  mm,	Y = 169.712  mm,	Z = -240.025  mm,
	W = 0.000 deg,	P = 30.000 deg,	R = 177.816 deg
};
P[295]{
   GP1:
	UF : 0, UT : 1,		CONFIG : 'N U T, 0, 0, 0',
	X = 1121.077  mm,	Y = 172.327  mm,	Z = -240.032  mm,
	W = 0.000 deg,	P = 30.000 deg,	R = 170.309 deg
};
P[296]{
   GP1:
	UF : 0, UT : 1,		CONFIG : 'N U T, 0, 0, 0',
	X = 1121.315  mm,	Y = 174.392  mm,	Z = -240.044  mm,
	W = 0.000 deg,	P = 30.000 deg,	R = 162.060 deg
};
P[297]{
   GP1:
	UF : 0, UT : 1,		CONFIG : 'N U T, 0, 0, 0',
	X = 1121.639  mm,	Y = 176.554  mm,	Z = -240.058  mm,
	W = 0.000 deg,	P = 30.000 deg,	R = 153.774 deg
};
P[298]{
   GP1:
	UF : 0, UT : 1,		CONFIG : 'N U T, 0, 0, 0',
	X = 1122.136  mm,	Y = 178.747  mm,	Z = -240.079  mm,
	W = 0.000 deg,	P = 30.000 deg,	R = 145.371 deg
};
P[299]{
   GP1:
	UF : 0, UT : 1,		CONFIG : 'N U T, 0, 0, 0',
	X = 1122.783  mm,	Y = 180.986  mm,	Z = -240.124  mm,
	W = 0.000 deg,	P = 30.000 deg,	R = 136.842 deg
};
P[300]{
   GP1:
	UF : 0, UT : 1,		CONFIG : 'N U T, 0, 0, 0',
	X = 1123.706  mm,	Y = 183.252  mm,	Z = -240.215  mm,
	W = 0.000 deg,	P = 30.000 deg,	R = 136.842 deg
};
P[301]{
   GP1:
	UF : 0, UT : 1,		CONFIG : 'N U T, 0, 0, 0',
	X = 1124.826  mm,	Y = 185.449  mm,	Z = -240.397  mm,
	W = 0.000 deg,	P = 30.000 deg,	R = 136.842 deg
};
P[302]{
   GP1:
	UF : 0, UT : 1,		CONFIG : 'N U T, 0, 0, 0',
	X = 1126.136  mm,	Y = 187.655  mm,	Z = -240.628  mm,
	W = 0.000 deg,	P = 30.000 deg,	R = 136.842 deg
};
P[303]{
   GP1:
	UF : 0, UT : 1,		CONFIG : 'N U T, 0, 0, 0',
	X = 1127.726  mm,	Y = 189.836  mm,	Z = -240.898  mm,
	W = 0.000 deg,	P = 30.000 deg,	R = 136.842 deg
};
P[304]{
   GP1:
	UF : 0, UT : 1,		CONFIG : 'N U T, 0, 0, 0',
	X = 1129.437  mm,	Y = 191.930  mm,	Z = -241.245  mm,
	W = 0.000 deg,	P = 30.000 deg,	R = 136.842 deg
};
P[305]{
   GP1:
	UF : 0, UT : 1,		CONFIG : 'N U T, 0, 0, 0',
	X = 1131.234  mm,	Y = 194.011  mm,	Z = -241.676  mm,
	W = 0.000 deg,	P = 30.000 deg,	R = 136.842 deg
};
P[306]{
   GP1:
	UF : 0, UT : 1,		CONFIG : 'N U T, 0, 0, 0',
	X = 1137.500  mm,	Y = 191.913  mm,	Z = -242.193  mm,
	W = 0.000 deg,	P = 30.000 deg,	R = 136.842 deg
};
P[307]{
   GP1:
	UF : 0, UT : 1,		CONFIG : 'N U T, 0, 0, 0',
	X = 1139.441  mm,	Y = 193.864  mm,	Z = -242.791  mm,
	W = 0.000 deg,	P = 30.000 deg,	R = 136.842 deg
};
P[308]{
   GP1:
	UF : 0, UT : 1,		CONFIG : 'N U T, 0, 0, 0',
	X = 1141.454  mm,	Y = 195.811  mm,	Z = -243.398  mm,
	W = 0.000 deg,	P = 30.000 deg,	R = 136.842 deg
};
P[309]{
   GP1:
	UF : 0, UT : 1,		CONFIG : 'N U T, 0, 0, 0',
	X = 1143.627  mm,	Y = 197.786  mm,	Z = -244.068  mm,
	W = 0.000 deg,	P = 30.000 deg,	R = 136.842 deg
};
P[310]{
   GP1:
	UF : 0, UT : 1,		CONFIG : 'N U T, 0, 0, 0',
	X = 1145.792  mm,	Y = 199.778  mm,	Z = -244.781  mm,
	W = 0.000 deg,	P = 30.000 deg,	R = 139.266 deg
};
P[311]{
   GP1:
	UF : 0, UT : 1,		CONFIG : 'N U T, 0, 0, 0',
	X = 1148.006  mm,	Y = 201.758  mm,	Z = -245.515  mm,
	W = 0.000 deg,	P = 30.000 deg,	R = 149.750 deg
};
P[312]{
   GP1:
	UF : 0, UT : 1,		CONFIG : 'N U T, 0, 0, 0',
	X = 1150.267  mm,	Y = 203.755  mm,	Z = -246.248  mm,
	W = 0.000 deg,	P = 30.000 deg,	R = 160.302 deg
};
P[313]{
   GP1:
	UF : 0, UT : 1,		CONFIG : 'N U T, 0, 0, 0',
	X = 1152.538  mm,	Y = 205.778  mm,	Z = -246.952  mm,
	W = 0.000 deg,	P = 30.000 deg,	R = 170.789 deg
};
P[314]{
   GP1:
	UF : 0, UT : 1,		CONFIG : 'N U T, 0, 0, 0',
	X = 1154.760  mm,	Y = 207.831  mm,	Z = -247.625  mm,
	W = 0.000 deg,	P = 30.000 deg,	R = 170.789 deg
};
P[315]{
   GP1:
	UF : 0, UT : 1,		CONFIG : 'N U T, 0, 0, 0',
	X = 1156.876  mm,	Y = 209.923  mm,	Z = -248.243  mm,
	W = 0.000 deg,	P = 30.000 deg,	R = 170.789 deg
};
P[316]{
   GP1:
	UF : 0, UT : 1,		CONFIG : 'N U T, 0, 0, 0',
	X = 1158.804  mm,	Y = 212.050  mm,	Z = -248.792  mm,
	W = 0.000 deg,	P = 30.000 deg,	R = 170.789 deg
};
P[317]{
   GP1:
	UF : 0, UT : 1,		CONFIG : 'N U T, 0, 0, 0',
	X = 1160.551  mm,	Y = 214.225  mm,	Z = -249.275  mm,
	W = 0.000 deg,	P = 30.000 deg,	R = 170.789 deg
};
P[318]{
   GP1:
	UF : 0, UT : 1,		CONFIG : 'N U T, 0, 0, 0',
	X = 1162.045  mm,	Y = 216.478  mm,	Z = -249.661  mm,
	W = 0.000 deg,	P = 30.000 deg,	R = 170.789 deg
};
P[319]{
   GP1:
	UF : 0, UT : 1,		CONFIG : 'N U T, 0, 0, 0',
	X = 1163.229  mm,	Y = 218.782  mm,	Z = -249.951  mm,
	W = 0.000 deg,	P = 30.000 deg,	R = 170.789 deg
};
P[320]{
   GP1:
	UF : 0, UT : 1,		CONFIG : 'N U T, 0, 0, 0',
	X = 1164.111  mm,	Y = 221.139  mm,	Z = -250.162  mm,
	W = 0.000 deg,	P = 30.000 deg,	R = 170.789 deg
};
P[321]{
   GP1:
	UF : 0, UT : 1,		CONFIG : 'N U T, 0, 0, 0',
	X = 1164.640  mm,	Y = 223.473  mm,	Z = -250.272  mm,
	W = 0.000 deg,	P = 30.000 deg,	R = 170.789 deg
};
P[322]{
   GP1:
	UF : 0, UT : 1,		CONFIG : 'N U T, 0, 0, 0',
	X = 1158.966  mm,	Y = 226.294  mm,	Z = -250.331  mm,
	W = 0.000 deg,	P = 30.000 deg,	R = 170.789 deg
};
P[323]{
   GP1:
	UF : 0, UT : 1,		CONFIG : 'N U T, 0, 0, 0',
	X = 1159.084  mm,	Y = 228.133  mm,	Z = -250.347  mm,
	W = 0.000 deg,	P = 30.000 deg,	R = 170.789 deg
};
P[324]{
   GP1:
	UF : 0, UT : 1,		CONFIG : 'N U T, 0, 0, 0',
	X = 1159.129  mm,	Y = 230.034  mm,	Z = -250.340  mm,
	W = 0.000 deg,	P = 30.000 deg,	R = 170.789 deg
};
P[325]{
   GP1:
	UF : 0, UT : 1,		CONFIG : 'N U T, 0, 0, 0',
	X = 1159.126  mm,	Y = 231.985  mm,	Z = -250.325  mm,
	W = 0.000 deg,	P = 30.000 deg,	R = 170.789 deg
};
P[326]{
   GP1:
	UF : 0, UT : 1,		CONFIG : 'N U T, 0, 0, 0',
	X = 1159.108  mm,	Y = 233.972  mm,	Z = -250.304  mm,
	W = 0.000 deg,	P = 30.000 deg,	R = 170.789 deg
};
P[327]{
   GP1:
	UF : 0, UT : 1,		CONFIG : 'N U T, 0, 0, 0',
	X = 1159.089  mm,	Y = 235.966  mm,	Z = -250.277  mm,
	W = 0.000 deg,	P = 30.000 deg,	R = 170.789 deg
};
P[328]{
   GP1:
	UF : 0, UT : 1,		CONFIG : 'N U T, 0, 0, 0',
	X = 1159.064  mm,	Y = 237.960  mm,	Z = -250.237  mm,
	W = 0.000 deg,	P = 30.000 deg,	R = 170.789 deg
};
P[329]{
   GP1:
	UF : 0, UT : 1,		CONFIG : 'N U T, 0, 0, 0',
	X = 1159.036  mm,	Y = 239.956  mm,	Z = -250.197  mm,
	W = 0.000 deg,	P = 30.000 deg,	R = 170.789 deg
};
P[330]{
   GP1:
	UF : 0, UT : 1,		CONFIG : 'N U T, 0, 0, 0',
	X = 1159.005  mm,	Y = 241.947  mm,	Z = -250.152  mm,
	W = 0.000 deg,	P = 30.000 deg,	R = 170.789 deg
};
P[331]{
   GP1:
	UF : 0, UT : 1,		CONFIG : 'N U T, 0, 0, 0',
	X = 1158.965  mm,	Y = 243.946  mm,	Z = -250.108  mm,
	W = 0.000 deg,	P = 30.000 deg,	R = 170.789 deg
};
P[332]{
   GP1:
	UF : 0, UT : 1,		CONFIG : 'N U T, 0, 0, 0',
	X = 1158.932  mm,	Y = 245.949  mm,	Z = -250.065  mm,
	W = 0.000 deg,	P = 30.000 deg,	R = 170.789 deg
};
P[333]{
   GP1:
	UF : 0, UT : 1,		CONFIG : 'N U T, 0, 0, 0',
	X = 1158.897  mm,	Y = 247.934  mm,	Z = -250.021  mm,
	W = 0.000 deg,	P = 30.000 deg,	R = 170.789 deg
};
P[334]{
   GP1:
	UF : 0, UT : 1,		CONFIG : 'N U T, 0, 0, 0',
	X = 1158.844  mm,	Y = 249.924  mm,	Z = -249.974  mm,
	W = 0.000 deg,	P = 30.000 deg,	R = 170.789 deg
};
P[335]{
   GP1:
	UF : 0, UT : 1,		CONFIG : 'N U T, 0, 0, 0',
	X = 1158.796  mm,	Y = 251.929  mm,	Z = -249.944  mm,
	W = 0.000 deg,	P = 30.000 deg,	R = 170.789 deg
};
P[336]{
   GP1:
	UF : 0, UT : 1,		CONFIG : 'N U T, 0, 0, 0',
	X = 1158.750  mm,	Y = 253.931  mm,	Z = -249.914  mm,
	W = 0.000 deg,	P = 30.000 deg,	R = 170.789 deg
};
/END
